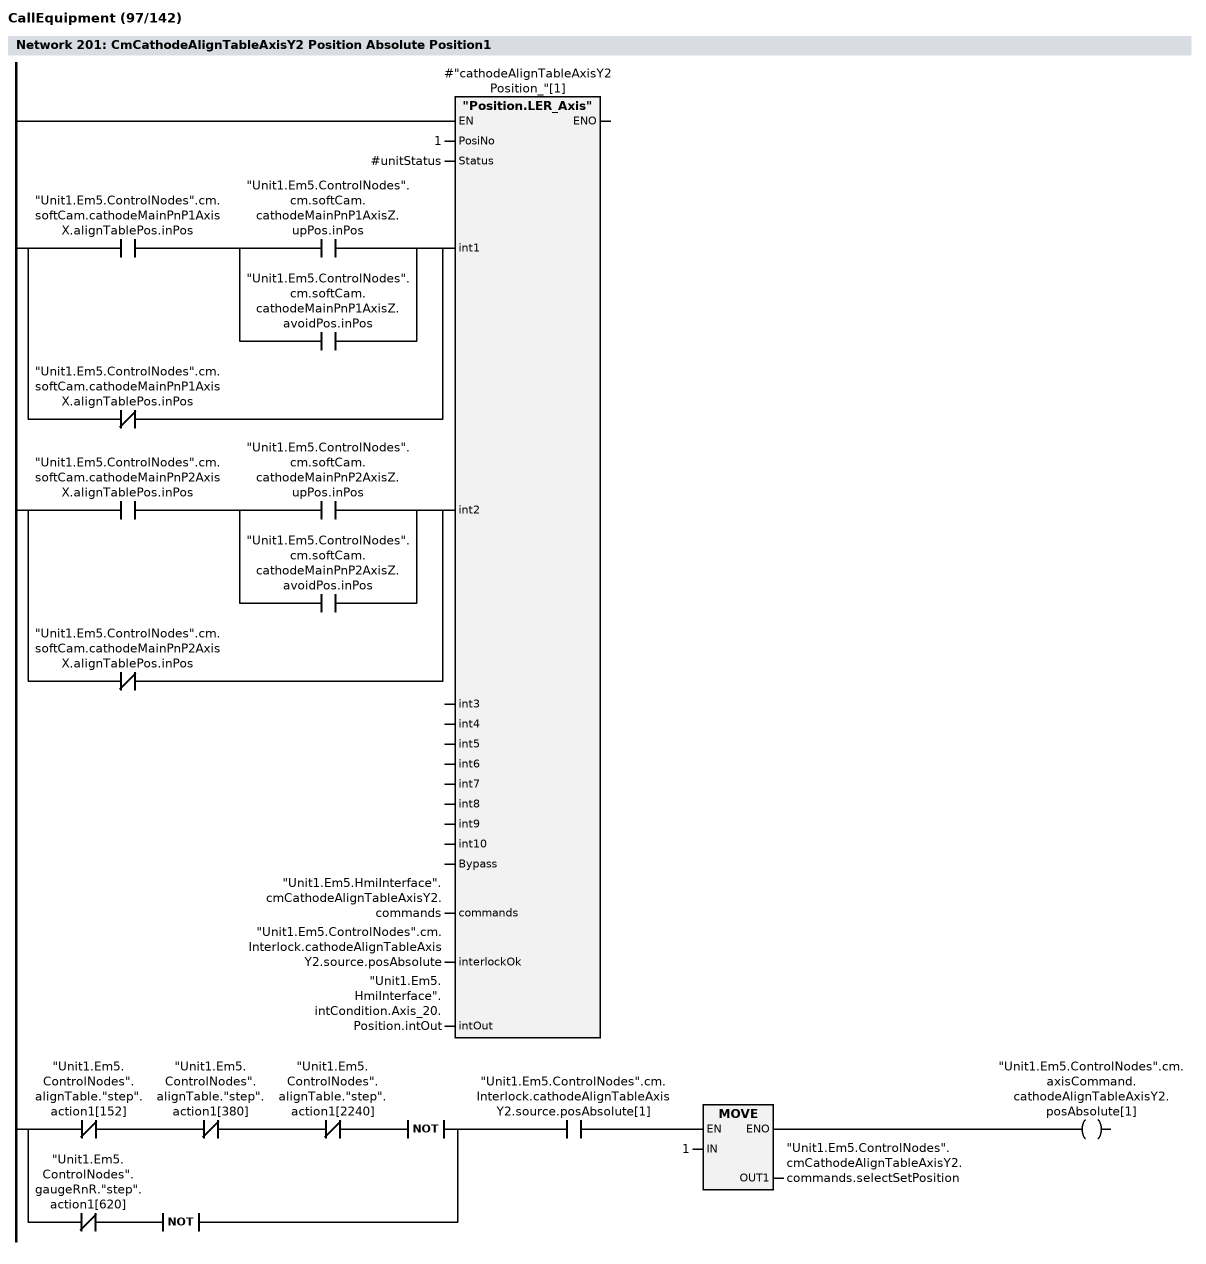
   RUNG wire#powerrail
      #"cathodeAlignTableAxisY2 Position_"[1](int1 := wire#w2, int2 := wire#w4, PosiNo := 1, Status := #unitStatus, int3 :=, int4 :=, int5 :=, int6 :=, int7 :=, int8 :=, int9 :=, int10 :=, Bypass :=, commands := "Unit1.Em5.HmiInterface".cmCathodeAlignTableAxisY2.commands, interlockOk := "Unit1.Em5.ControlNodes".cm.Interlock.cathodeAlignTableAxisY2.source.posAbsolute, intOut := "Unit1.Em5.HmiInterface".intCondition.Axis_20.Position.intOut)
   END_RUNG
   RUNG wire#powerrail
      Contact( "Unit1.Em5.ControlNodes".cm.softCam.cathodeMainPnP1AxisX.alignTablePos.inPos )
      wire#w1
      Contact( "Unit1.Em5.ControlNodes".cm.softCam.cathodeMainPnP1AxisZ.upPos.inPos )
   END_RUNG wire#w2
   RUNG wire#w1
      Contact( "Unit1.Em5.ControlNodes".cm.softCam.cathodeMainPnP1AxisZ.avoidPos.inPos )
   END_RUNG wire#w2
   RUNG wire#powerrail
      I_Contact( "Unit1.Em5.ControlNodes".cm.softCam.cathodeMainPnP1AxisX.alignTablePos.inPos )
   END_RUNG wire#w2
   RUNG wire#powerrail
      Contact( "Unit1.Em5.ControlNodes".cm.softCam.cathodeMainPnP2AxisX.alignTablePos.inPos )
      wire#w3
      Contact( "Unit1.Em5.ControlNodes".cm.softCam.cathodeMainPnP2AxisZ.upPos.inPos )
   END_RUNG wire#w4
   RUNG wire#w3
      Contact( "Unit1.Em5.ControlNodes".cm.softCam.cathodeMainPnP2AxisZ.avoidPos.inPos )
   END_RUNG wire#w4
   RUNG wire#powerrail
      I_Contact( "Unit1.Em5.ControlNodes".cm.softCam.cathodeMainPnP2AxisX.alignTablePos.inPos )
   END_RUNG wire#w4
   RUNG wire#powerrail
      I_Contact( "Unit1.Em5.ControlNodes".alignTable."step".action1[152] )
      I_Contact( "Unit1.Em5.ControlNodes".alignTable."step".action1[380] )
      I_Contact( "Unit1.Em5.ControlNodes".alignTable."step".action1[2240] )
      Not()
      wire#w5
      Contact( "Unit1.Em5.ControlNodes".cm.Interlock.cathodeAlignTableAxisY2.source.posAbsolute[1] )
      Move(in := 1, out1 => "Unit1.Em5.ControlNodes".cmCathodeAlignTableAxisY2.commands.selectSetPosition)
      Coil( "Unit1.Em5.ControlNodes".cm.axisCommand.cathodeAlignTableAxisY2.posAbsolute[1] )
   END_RUNG
   RUNG wire#powerrail
      I_Contact( "Unit1.Em5.ControlNodes".gaugeRnR."step".action1[620] )
      Not()
   END_RUNG wire#w5
   // the same network as SCL:
   #"cathodeAlignTableAxisY2 Position_"[1](PosiNo := 1,   // "Position.LER_Axis"
                           Status := #unitStatus,
                           int1 := ("Unit1.Em5.ControlNodes".cm.softCam.cathodeMainPnP1AxisX.alignTablePos.inPos AND ("Unit1.Em5.ControlNodes".cm.softCam.cathodeMainPnP1AxisZ.upPos.inPos OR "Unit1.Em5.ControlNodes".cm.softCam.cathodeMainPnP1AxisZ.avoidPos.inPos)) OR NOT "Unit1.Em5.ControlNodes".cm.softCam.cathodeMainPnP1AxisX.alignTablePos.inPos,
                           int2 := ("Unit1.Em5.ControlNodes".cm.softCam.cathodeMainPnP2AxisX.alignTablePos.inPos AND ("Unit1.Em5.ControlNodes".cm.softCam.cathodeMainPnP2AxisZ.upPos.inPos OR "Unit1.Em5.ControlNodes".cm.softCam.cathodeMainPnP2AxisZ.avoidPos.inPos)) OR NOT "Unit1.Em5.ControlNodes".cm.softCam.cathodeMainPnP2AxisX.alignTablePos.inPos,
                           commands := "Unit1.Em5.HmiInterface".cmCathodeAlignTableAxisY2.commands,
                           interlockOk := "Unit1.Em5.ControlNodes".cm.Interlock.cathodeAlignTableAxisY2.source.posAbsolute,
                           intOut := "Unit1.Em5.HmiInterface".intCondition.Axis_20.Position.intOut);
   #_w1 := (NOT (NOT "Unit1.Em5.ControlNodes".alignTable."step".action1[152] AND NOT "Unit1.Em5.ControlNodes".alignTable."step".action1[380] AND NOT "Unit1.Em5.ControlNodes".alignTable."step".action1[2240]) OR NOT (NOT "Unit1.Em5.ControlNodes".gaugeRnR."step".action1[620])) AND "Unit1.Em5.ControlNodes".cm.Interlock.cathodeAlignTableAxisY2.source.posAbsolute[1];
   IF #_w1 THEN "Unit1.Em5.ControlNodes".cmCathodeAlignTableAxisY2.commands.selectSetPosition := 1; END_IF;
   "Unit1.Em5.ControlNodes".cm.axisCommand.cathodeAlignTableAxisY2.posAbsolute[1] := #_w1;
END_REGION

REGION Network 202: CmCathodeAlignTableAxisY2 Position Absolute Position2
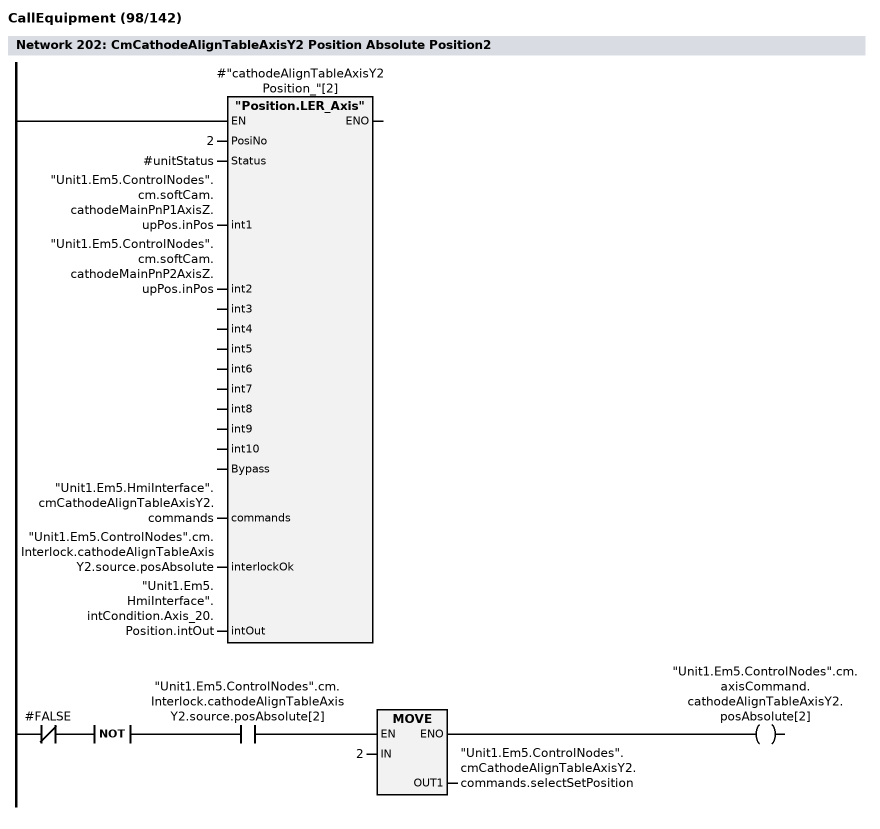
   RUNG wire#powerrail
      #"cathodeAlignTableAxisY2 Position_"[2](PosiNo := 2, Status := #unitStatus, int1 := "Unit1.Em5.ControlNodes".cm.softCam.cathodeMainPnP1AxisZ.upPos.inPos, int2 := "Unit1.Em5.ControlNodes".cm.softCam.cathodeMainPnP2AxisZ.upPos.inPos, int3 :=, int4 :=, int5 :=, int6 :=, int7 :=, int8 :=, int9 :=, int10 :=, Bypass :=, commands := "Unit1.Em5.HmiInterface".cmCathodeAlignTableAxisY2.commands, interlockOk := "Unit1.Em5.ControlNodes".cm.Interlock.cathodeAlignTableAxisY2.source.posAbsolute, intOut := "Unit1.Em5.HmiInterface".intCondition.Axis_20.Position.intOut)
   END_RUNG
   RUNG wire#powerrail
      I_Contact( #FALSE )
      Not()
      Contact( "Unit1.Em5.ControlNodes".cm.Interlock.cathodeAlignTableAxisY2.source.posAbsolute[2] )
      Move(in := 2, out1 => "Unit1.Em5.ControlNodes".cmCathodeAlignTableAxisY2.commands.selectSetPosition)
      Coil( "Unit1.Em5.ControlNodes".cm.axisCommand.cathodeAlignTableAxisY2.posAbsolute[2] )
   END_RUNG
   // the same network as SCL:
   #"cathodeAlignTableAxisY2 Position_"[2](PosiNo := 2,   // "Position.LER_Axis"
                           Status := #unitStatus,
                           int1 := "Unit1.Em5.ControlNodes".cm.softCam.cathodeMainPnP1AxisZ.upPos.inPos,
                           int2 := "Unit1.Em5.ControlNodes".cm.softCam.cathodeMainPnP2AxisZ.upPos.inPos,
                           commands := "Unit1.Em5.HmiInterface".cmCathodeAlignTableAxisY2.commands,
                           interlockOk := "Unit1.Em5.ControlNodes".cm.Interlock.cathodeAlignTableAxisY2.source.posAbsolute,
                           intOut := "Unit1.Em5.HmiInterface".intCondition.Axis_20.Position.intOut);
   #_w1 := NOT (NOT #FALSE) AND "Unit1.Em5.ControlNodes".cm.Interlock.cathodeAlignTableAxisY2.source.posAbsolute[2];
   IF #_w1 THEN "Unit1.Em5.ControlNodes".cmCathodeAlignTableAxisY2.commands.selectSetPosition := 2; END_IF;
   "Unit1.Em5.ControlNodes".cm.axisCommand.cathodeAlignTableAxisY2.posAbsolute[2] := #_w1;
END_REGION

REGION Network 203: CmCathodeAlignTableAxisY2 Position Absolute Position3
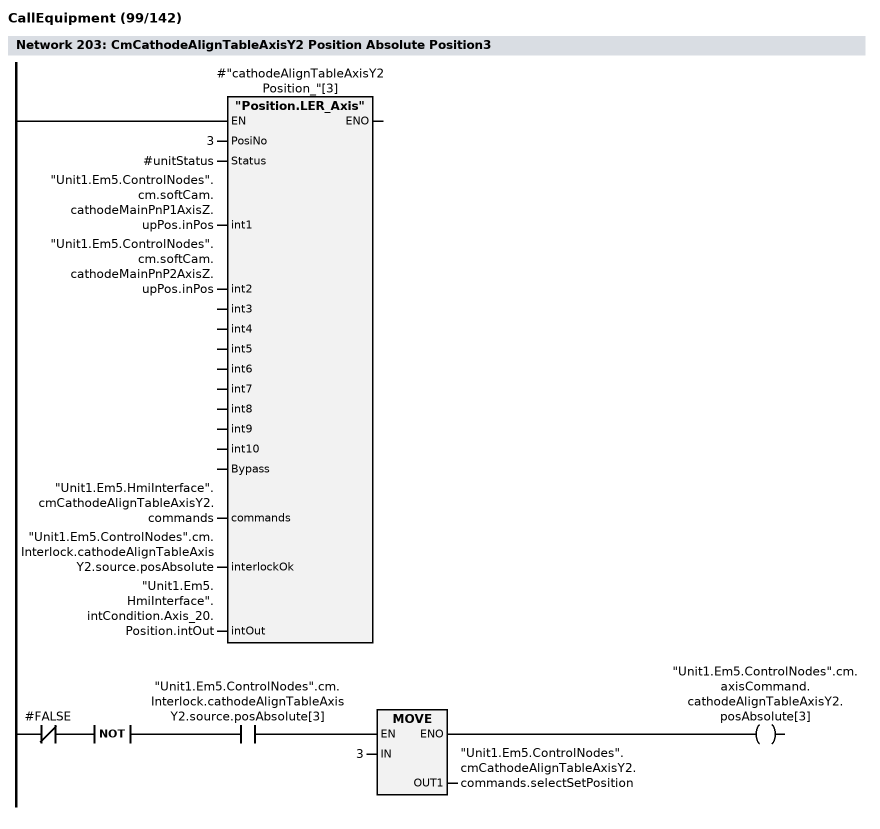
   RUNG wire#powerrail
      #"cathodeAlignTableAxisY2 Position_"[3](PosiNo := 3, Status := #unitStatus, int1 := "Unit1.Em5.ControlNodes".cm.softCam.cathodeMainPnP1AxisZ.upPos.inPos, int2 := "Unit1.Em5.ControlNodes".cm.softCam.cathodeMainPnP2AxisZ.upPos.inPos, int3 :=, int4 :=, int5 :=, int6 :=, int7 :=, int8 :=, int9 :=, int10 :=, Bypass :=, commands := "Unit1.Em5.HmiInterface".cmCathodeAlignTableAxisY2.commands, interlockOk := "Unit1.Em5.ControlNodes".cm.Interlock.cathodeAlignTableAxisY2.source.posAbsolute, intOut := "Unit1.Em5.HmiInterface".intCondition.Axis_20.Position.intOut)
   END_RUNG
   RUNG wire#powerrail
      I_Contact( #FALSE )
      Not()
      Contact( "Unit1.Em5.ControlNodes".cm.Interlock.cathodeAlignTableAxisY2.source.posAbsolute[3] )
      Move(in := 3, out1 => "Unit1.Em5.ControlNodes".cmCathodeAlignTableAxisY2.commands.selectSetPosition)
      Coil( "Unit1.Em5.ControlNodes".cm.axisCommand.cathodeAlignTableAxisY2.posAbsolute[3] )
   END_RUNG
   // the same network as SCL:
   #"cathodeAlignTableAxisY2 Position_"[3](PosiNo := 3,   // "Position.LER_Axis"
                           Status := #unitStatus,
                           int1 := "Unit1.Em5.ControlNodes".cm.softCam.cathodeMainPnP1AxisZ.upPos.inPos,
                           int2 := "Unit1.Em5.ControlNodes".cm.softCam.cathodeMainPnP2AxisZ.upPos.inPos,
                           commands := "Unit1.Em5.HmiInterface".cmCathodeAlignTableAxisY2.commands,
                           interlockOk := "Unit1.Em5.ControlNodes".cm.Interlock.cathodeAlignTableAxisY2.source.posAbsolute,
                           intOut := "Unit1.Em5.HmiInterface".intCondition.Axis_20.Position.intOut);
   #_w1 := NOT (NOT #FALSE) AND "Unit1.Em5.ControlNodes".cm.Interlock.cathodeAlignTableAxisY2.source.posAbsolute[3];
   IF #_w1 THEN "Unit1.Em5.ControlNodes".cmCathodeAlignTableAxisY2.commands.selectSetPosition := 3; END_IF;
   "Unit1.Em5.ControlNodes".cm.axisCommand.cathodeAlignTableAxisY2.posAbsolute[3] := #_w1;
END_REGION

REGION Network 204: CmCathodeAlignTableAxisY2 Position Absolute Position4
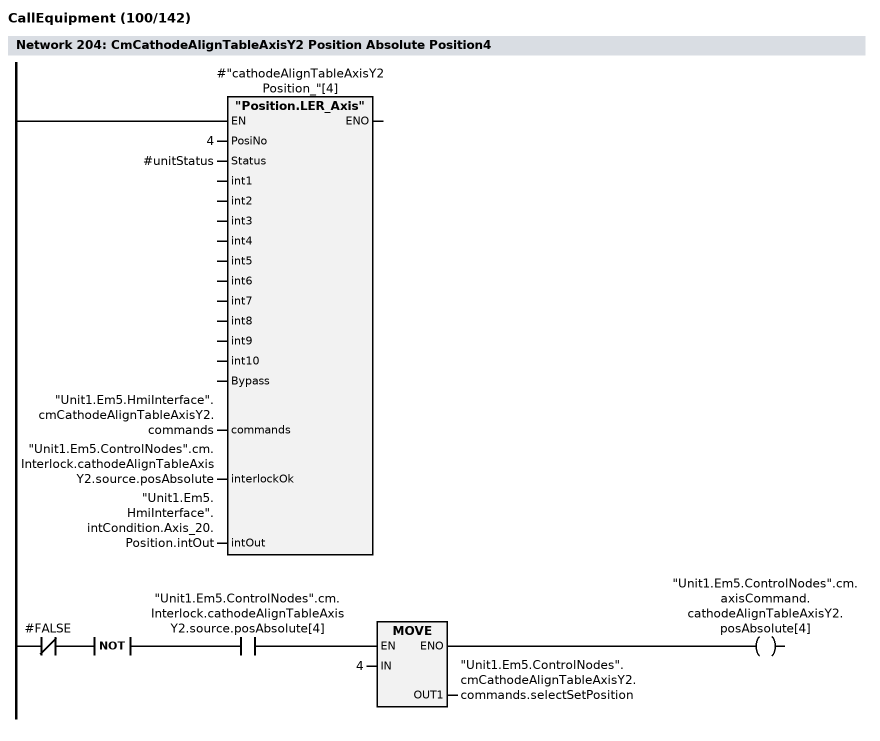
   RUNG wire#powerrail
      #"cathodeAlignTableAxisY2 Position_"[4](PosiNo := 4, Status := #unitStatus, int1 :=, int2 :=, int3 :=, int4 :=, int5 :=, int6 :=, int7 :=, int8 :=, int9 :=, int10 :=, Bypass :=, commands := "Unit1.Em5.HmiInterface".cmCathodeAlignTableAxisY2.commands, interlockOk := "Unit1.Em5.ControlNodes".cm.Interlock.cathodeAlignTableAxisY2.source.posAbsolute, intOut := "Unit1.Em5.HmiInterface".intCondition.Axis_20.Position.intOut)
   END_RUNG
   RUNG wire#powerrail
      I_Contact( #FALSE )
      Not()
      Contact( "Unit1.Em5.ControlNodes".cm.Interlock.cathodeAlignTableAxisY2.source.posAbsolute[4] )
      Move(in := 4, out1 => "Unit1.Em5.ControlNodes".cmCathodeAlignTableAxisY2.commands.selectSetPosition)
      Coil( "Unit1.Em5.ControlNodes".cm.axisCommand.cathodeAlignTableAxisY2.posAbsolute[4] )
   END_RUNG
   // the same network as SCL:
   #"cathodeAlignTableAxisY2 Position_"[4](PosiNo := 4,   // "Position.LER_Axis"
                           Status := #unitStatus,
                           commands := "Unit1.Em5.HmiInterface".cmCathodeAlignTableAxisY2.commands,
                           interlockOk := "Unit1.Em5.ControlNodes".cm.Interlock.cathodeAlignTableAxisY2.source.posAbsolute,
                           intOut := "Unit1.Em5.HmiInterface".intCondition.Axis_20.Position.intOut);
   #_w1 := NOT (NOT #FALSE) AND "Unit1.Em5.ControlNodes".cm.Interlock.cathodeAlignTableAxisY2.source.posAbsolute[4];
   IF #_w1 THEN "Unit1.Em5.ControlNodes".cmCathodeAlignTableAxisY2.commands.selectSetPosition := 4; END_IF;
   "Unit1.Em5.ControlNodes".cm.axisCommand.cathodeAlignTableAxisY2.posAbsolute[4] := #_w1;
END_REGION

REGION Network 205: CmCathodeAlignTableAxisY2 Position Absolute Position5
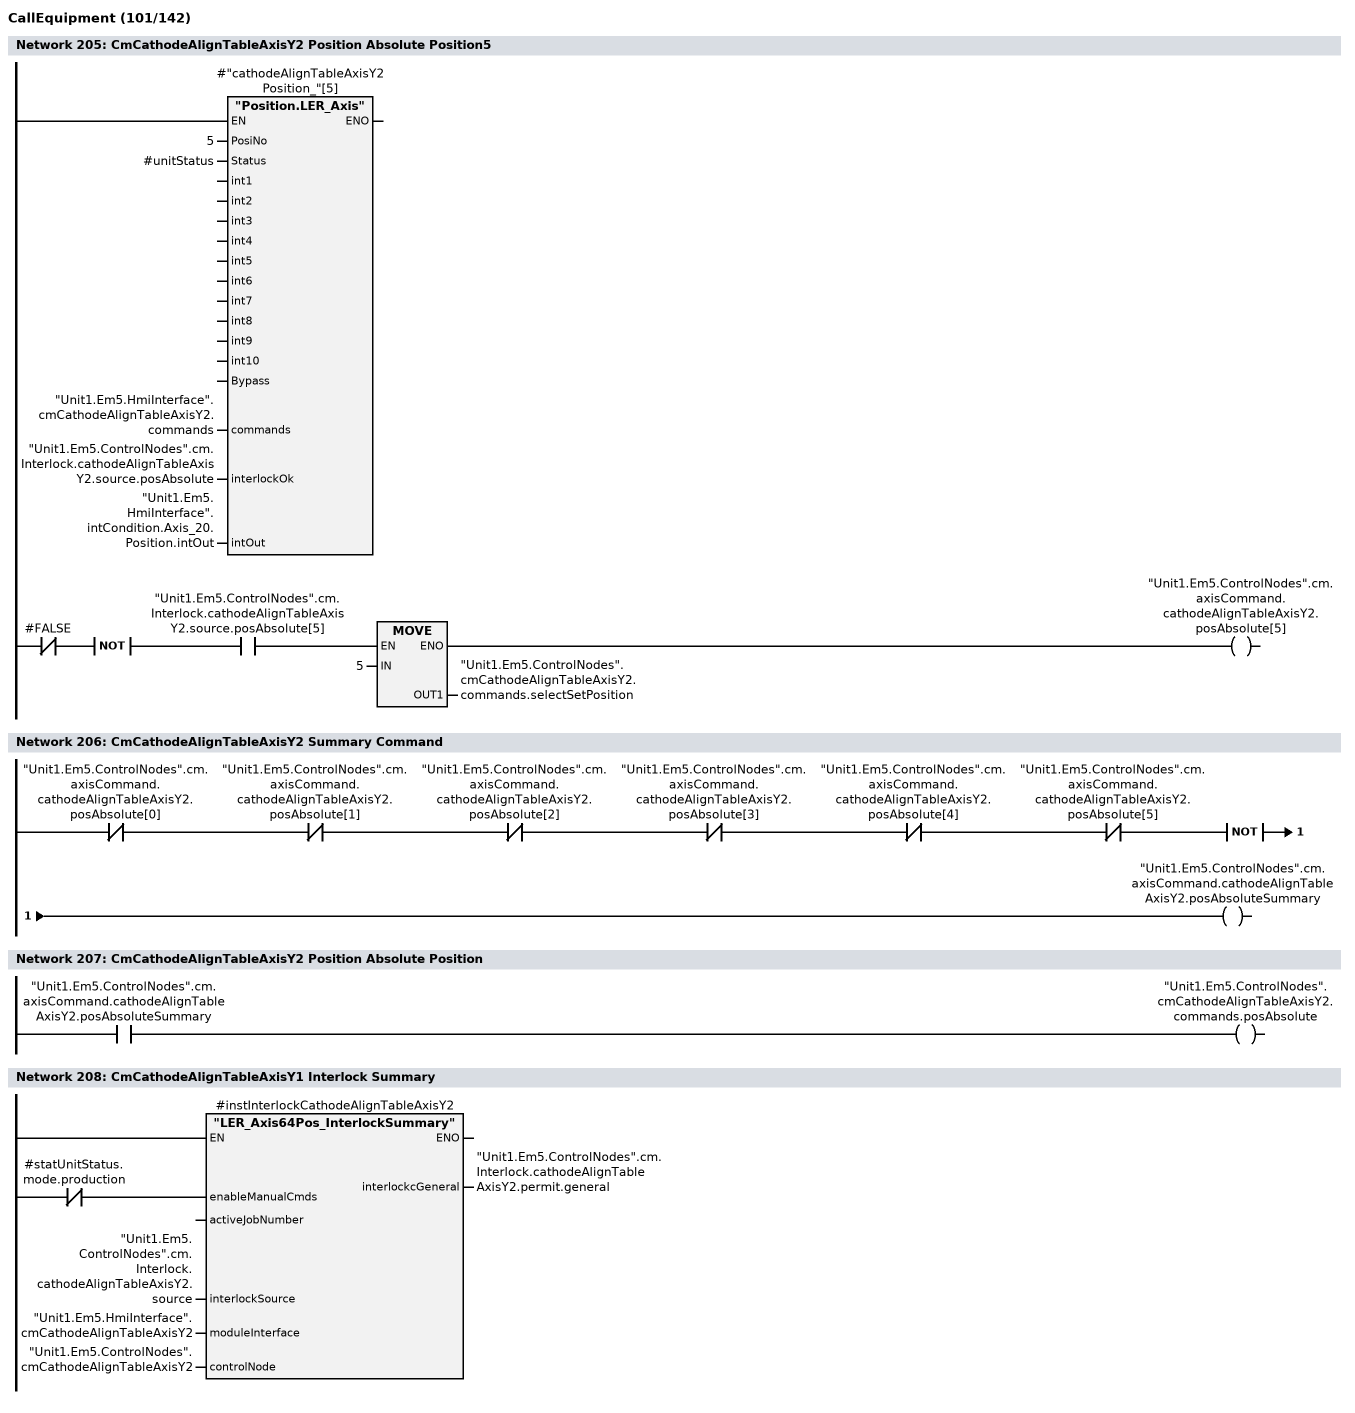
   RUNG wire#powerrail
      #"cathodeAlignTableAxisY2 Position_"[5](PosiNo := 5, Status := #unitStatus, int1 :=, int2 :=, int3 :=, int4 :=, int5 :=, int6 :=, int7 :=, int8 :=, int9 :=, int10 :=, Bypass :=, commands := "Unit1.Em5.HmiInterface".cmCathodeAlignTableAxisY2.commands, interlockOk := "Unit1.Em5.ControlNodes".cm.Interlock.cathodeAlignTableAxisY2.source.posAbsolute, intOut := "Unit1.Em5.HmiInterface".intCondition.Axis_20.Position.intOut)
   END_RUNG
   RUNG wire#powerrail
      I_Contact( #FALSE )
      Not()
      Contact( "Unit1.Em5.ControlNodes".cm.Interlock.cathodeAlignTableAxisY2.source.posAbsolute[5] )
      Move(in := 5, out1 => "Unit1.Em5.ControlNodes".cmCathodeAlignTableAxisY2.commands.selectSetPosition)
      Coil( "Unit1.Em5.ControlNodes".cm.axisCommand.cathodeAlignTableAxisY2.posAbsolute[5] )
   END_RUNG
   // the same network as SCL:
   #"cathodeAlignTableAxisY2 Position_"[5](PosiNo := 5,   // "Position.LER_Axis"
                           Status := #unitStatus,
                           commands := "Unit1.Em5.HmiInterface".cmCathodeAlignTableAxisY2.commands,
                           interlockOk := "Unit1.Em5.ControlNodes".cm.Interlock.cathodeAlignTableAxisY2.source.posAbsolute,
                           intOut := "Unit1.Em5.HmiInterface".intCondition.Axis_20.Position.intOut);
   #_w1 := NOT (NOT #FALSE) AND "Unit1.Em5.ControlNodes".cm.Interlock.cathodeAlignTableAxisY2.source.posAbsolute[5];
   IF #_w1 THEN "Unit1.Em5.ControlNodes".cmCathodeAlignTableAxisY2.commands.selectSetPosition := 5; END_IF;
   "Unit1.Em5.ControlNodes".cm.axisCommand.cathodeAlignTableAxisY2.posAbsolute[5] := #_w1;
END_REGION

REGION Network 206: CmCathodeAlignTableAxisY2 Summary Command
   RUNG wire#powerrail
      I_Contact( "Unit1.Em5.ControlNodes".cm.axisCommand.cathodeAlignTableAxisY2.posAbsolute[0] )
      I_Contact( "Unit1.Em5.ControlNodes".cm.axisCommand.cathodeAlignTableAxisY2.posAbsolute[1] )
      I_Contact( "Unit1.Em5.ControlNodes".cm.axisCommand.cathodeAlignTableAxisY2.posAbsolute[2] )
      I_Contact( "Unit1.Em5.ControlNodes".cm.axisCommand.cathodeAlignTableAxisY2.posAbsolute[3] )
      I_Contact( "Unit1.Em5.ControlNodes".cm.axisCommand.cathodeAlignTableAxisY2.posAbsolute[4] )
      I_Contact( "Unit1.Em5.ControlNodes".cm.axisCommand.cathodeAlignTableAxisY2.posAbsolute[5] )
      Not()
      Coil( "Unit1.Em5.ControlNodes".cm.axisCommand.cathodeAlignTableAxisY2.posAbsoluteSummary )
   END_RUNG
   // the same network as SCL:
   "Unit1.Em5.ControlNodes".cm.axisCommand.cathodeAlignTableAxisY2.posAbsoluteSummary := NOT (NOT "Unit1.Em5.ControlNodes".cm.axisCommand.cathodeAlignTableAxisY2.posAbsolute[0] AND NOT "Unit1.Em5.ControlNodes".cm.axisCommand.cathodeAlignTableAxisY2.posAbsolute[1] AND NOT "Unit1.Em5.ControlNodes".cm.axisCommand.cathodeAlignTableAxisY2.posAbsolute[2] AND NOT "Unit1.Em5.ControlNodes".cm.axisCommand.cathodeAlignTableAxisY2.posAbsolute[3] AND NOT "Unit1.Em5.ControlNodes".cm.axisCommand.cathodeAlignTableAxisY2.posAbsolute[4] AND NOT "Unit1.Em5.ControlNodes".cm.axisCommand.cathodeAlignTableAxisY2.posAbsolute[5]);
END_REGION

REGION Network 207: CmCathodeAlignTableAxisY2 Position Absolute Position
   RUNG wire#powerrail
      Contact( "Unit1.Em5.ControlNodes".cm.axisCommand.cathodeAlignTableAxisY2.posAbsoluteSummary )
      Coil( "Unit1.Em5.ControlNodes".cmCathodeAlignTableAxisY2.commands.posAbsolute )
   END_RUNG
   // the same network as SCL:
   "Unit1.Em5.ControlNodes".cmCathodeAlignTableAxisY2.commands.posAbsolute := "Unit1.Em5.ControlNodes".cm.axisCommand.cathodeAlignTableAxisY2.posAbsoluteSummary;
END_REGION

REGION Network 208: CmCathodeAlignTableAxisY1 Interlock Summary
   RUNG wire#powerrail
      #instInterlockCathodeAlignTableAxisY2(enableManualCmds := wire#w1, activeJobNumber :=, interlockSource := "Unit1.Em5.ControlNodes".cm.Interlock.cathodeAlignTableAxisY2.source, moduleInterface := "Unit1.Em5.HmiInterface".cmCathodeAlignTableAxisY2, controlNode := "Unit1.Em5.ControlNodes".cmCathodeAlignTableAxisY2, interlockcGeneral => "Unit1.Em5.ControlNodes".cm.Interlock.cathodeAlignTableAxisY2.permit.general)
   END_RUNG
   RUNG wire#powerrail
      I_Contact( #statUnitStatus.mode.production )
   END_RUNG wire#w1
   // the same network as SCL:
   #instInterlockCathodeAlignTableAxisY2(enableManualCmds := NOT #statUnitStatus.mode.production,   // "LER_Axis64Pos_InterlockSummary"
                           interlockSource := "Unit1.Em5.ControlNodes".cm.Interlock.cathodeAlignTableAxisY2.source,
                           moduleInterface := "Unit1.Em5.HmiInterface".cmCathodeAlignTableAxisY2,
                           controlNode := "Unit1.Em5.ControlNodes".cmCathodeAlignTableAxisY2,
                           interlockcGeneral => "Unit1.Em5.ControlNodes".cm.Interlock.cathodeAlignTableAxisY2.permit.general);
END_REGION

REGION Network 209: CmCathodeAlignTableAxisY2 velocity/speed
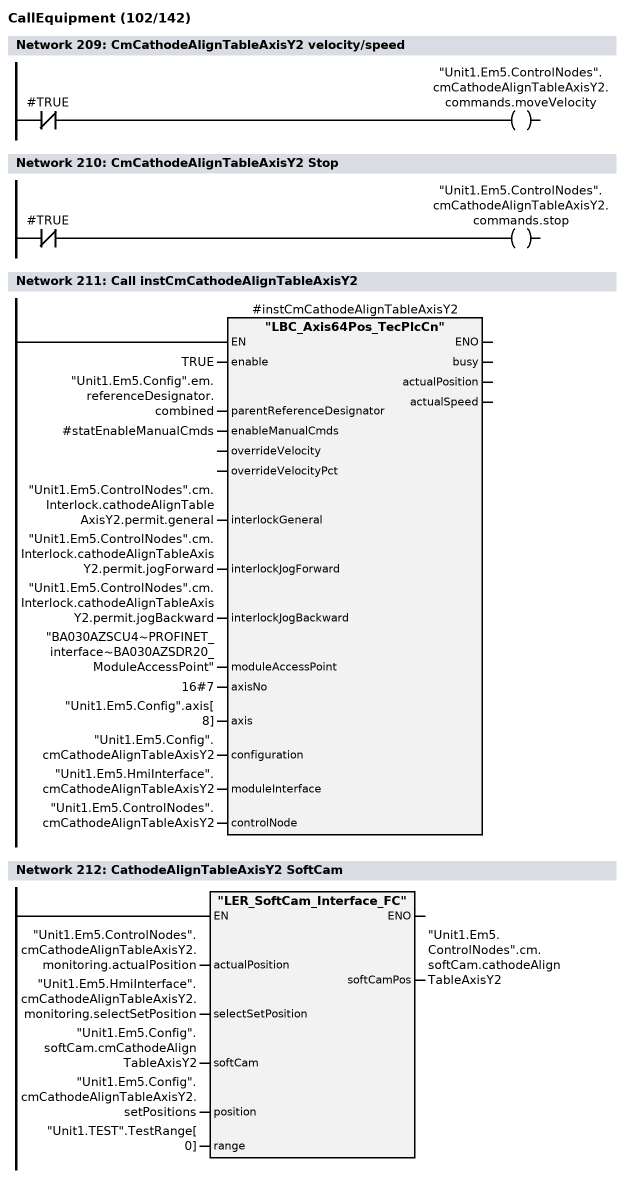
   RUNG wire#powerrail
      I_Contact( #TRUE )
      Coil( "Unit1.Em5.ControlNodes".cmCathodeAlignTableAxisY2.commands.moveVelocity )
   END_RUNG
   // the same network as SCL:
   "Unit1.Em5.ControlNodes".cmCathodeAlignTableAxisY2.commands.moveVelocity := NOT #TRUE;
END_REGION

REGION Network 210: CmCathodeAlignTableAxisY2 Stop
   RUNG wire#powerrail
      I_Contact( #TRUE )
      Coil( "Unit1.Em5.ControlNodes".cmCathodeAlignTableAxisY2.commands.stop )
   END_RUNG
   // the same network as SCL:
   "Unit1.Em5.ControlNodes".cmCathodeAlignTableAxisY2.commands.stop := NOT #TRUE;
END_REGION

REGION Network 211: Call instCmCathodeAlignTableAxisY2
   RUNG wire#powerrail
      #instCmCathodeAlignTableAxisY2(enable := TRUE, parentReferenceDesignator := "Unit1.Em5.Config".em.referenceDesignator.combined, enableManualCmds := #statEnableManualCmds, overrideVelocity :=, overrideVelocityPct :=, interlockGeneral := "Unit1.Em5.ControlNodes".cm.Interlock.cathodeAlignTableAxisY2.permit.general, interlockJogForward := "Unit1.Em5.ControlNodes".cm.Interlock.cathodeAlignTableAxisY2.permit.jogForward, interlockJogBackward := "Unit1.Em5.ControlNodes".cm.Interlock.cathodeAlignTableAxisY2.permit.jogBackward, moduleAccessPoint := "BA030AZSCU4~PROFINET_interface~BA030AZSDR20_ModuleAccessPoint", axisNo := 16#7, axis := "Unit1.Em5.Config".axis[8], configuration := "Unit1.Em5.Config".cmCathodeAlignTableAxisY2, moduleInterface := "Unit1.Em5.HmiInterface".cmCathodeAlignTableAxisY2, controlNode := "Unit1.Em5.ControlNodes".cmCathodeAlignTableAxisY2, busy =>, actualPosition =>, actualSpeed =>)
   END_RUNG
   // the same network as SCL:
   #instCmCathodeAlignTableAxisY2(enable := TRUE,   // "LBC_Axis64Pos_TecPlcCn"
                           parentReferenceDesignator := "Unit1.Em5.Config".em.referenceDesignator.combined,
                           enableManualCmds := #statEnableManualCmds,
                           interlockGeneral := "Unit1.Em5.ControlNodes".cm.Interlock.cathodeAlignTableAxisY2.permit.general,
                           interlockJogForward := "Unit1.Em5.ControlNodes".cm.Interlock.cathodeAlignTableAxisY2.permit.jogForward,
                           interlockJogBackward := "Unit1.Em5.ControlNodes".cm.Interlock.cathodeAlignTableAxisY2.permit.jogBackward,
                           moduleAccessPoint := "BA030AZSCU4~PROFINET_interface~BA030AZSDR20_ModuleAccessPoint",
                           axisNo := 16#7,
                           axis := "Unit1.Em5.Config".axis[8],
                           configuration := "Unit1.Em5.Config".cmCathodeAlignTableAxisY2,
                           moduleInterface := "Unit1.Em5.HmiInterface".cmCathodeAlignTableAxisY2,
                           controlNode := "Unit1.Em5.ControlNodes".cmCathodeAlignTableAxisY2);
END_REGION

REGION Network 212: CathodeAlignTableAxisY2 SoftCam
   RUNG wire#powerrail
      "LER_SoftCam_Interface_FC"(actualPosition := "Unit1.Em5.ControlNodes".cmCathodeAlignTableAxisY2.monitoring.actualPosition, selectSetPosition := "Unit1.Em5.HmiInterface".cmCathodeAlignTableAxisY2.monitoring.selectSetPosition, softCam := "Unit1.Em5.Config".softCam.cmCathodeAlignTableAxisY2, position := "Unit1.Em5.Config".cmCathodeAlignTableAxisY2.setPositions, range := "Unit1.TEST".TestRange[0], softCamPos => "Unit1.Em5.ControlNodes".cm.softCam.cathodeAlignTableAxisY2)
   END_RUNG
   // the same network as SCL:
   "LER_SoftCam_Interface_FC"(actualPosition := "Unit1.Em5.ControlNodes".cmCathodeAlignTableAxisY2.monitoring.actualPosition,
                           selectSetPosition := "Unit1.Em5.HmiInterface".cmCathodeAlignTableAxisY2.monitoring.selectSetPosition,
                           softCam := "Unit1.Em5.Config".softCam.cmCathodeAlignTableAxisY2,
                           position := "Unit1.Em5.Config".cmCathodeAlignTableAxisY2.setPositions,
                           range := "Unit1.TEST".TestRange[0],
                           softCamPos => "Unit1.Em5.ControlNodes".cm.softCam.cathodeAlignTableAxisY2);
END_REGION

REGION Network 213: ******************** Brake Test (Axis) ********************
END_REGION

REGION Network 214: Cathode Main PnP 1 Z-Axis Brake Test
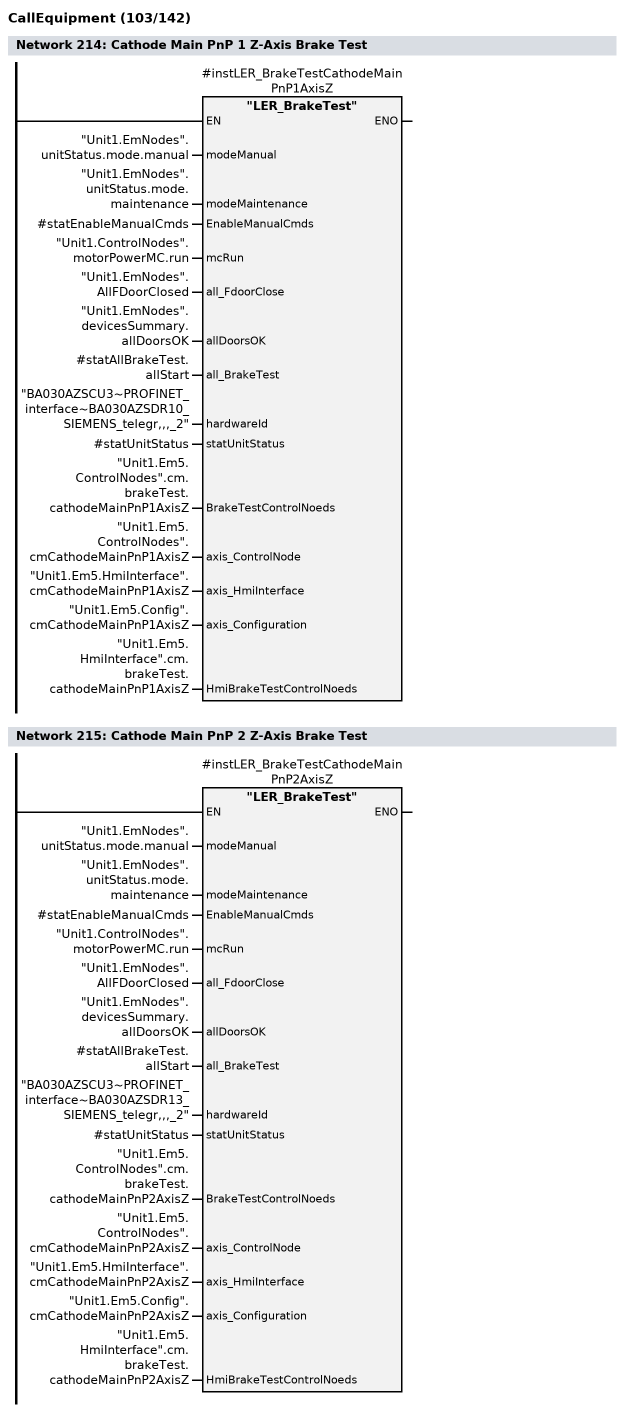
   RUNG wire#powerrail
      #instLER_BrakeTestCathodeMainPnP1AxisZ(modeManual := "Unit1.EmNodes".unitStatus.mode.manual, modeMaintenance := "Unit1.EmNodes".unitStatus.mode.maintenance, EnableManualCmds := #statEnableManualCmds, mcRun := "Unit1.ControlNodes".motorPowerMC.run, all_FdoorClose := "Unit1.EmNodes".AllFDoorClosed, allDoorsOK := "Unit1.EmNodes".devicesSummary.allDoorsOK, all_BrakeTest := #statAllBrakeTest.allStart, hardwareId := "BA030AZSCU3~PROFINET_interface~BA030AZSDR10_SIEMENS_telegr,,,_2", statUnitStatus := #statUnitStatus, BrakeTestControlNoeds := "Unit1.Em5.ControlNodes".cm.brakeTest.cathodeMainPnP1AxisZ, axis_ControlNode := "Unit1.Em5.ControlNodes".cmCathodeMainPnP1AxisZ, axis_HmiInterface := "Unit1.Em5.HmiInterface".cmCathodeMainPnP1AxisZ, axis_Configuration := "Unit1.Em5.Config".cmCathodeMainPnP1AxisZ, HmiBrakeTestControlNoeds := "Unit1.Em5.HmiInterface".cm.brakeTest.cathodeMainPnP1AxisZ)
   END_RUNG
   // the same network as SCL:
   #instLER_BrakeTestCathodeMainPnP1AxisZ(modeManual := "Unit1.EmNodes".unitStatus.mode.manual,   // "LER_BrakeTest"
                           modeMaintenance := "Unit1.EmNodes".unitStatus.mode.maintenance,
                           EnableManualCmds := #statEnableManualCmds,
                           mcRun := "Unit1.ControlNodes".motorPowerMC.run,
                           all_FdoorClose := "Unit1.EmNodes".AllFDoorClosed,
                           allDoorsOK := "Unit1.EmNodes".devicesSummary.allDoorsOK,
                           all_BrakeTest := #statAllBrakeTest.allStart,
                           hardwareId := "BA030AZSCU3~PROFINET_interface~BA030AZSDR10_SIEMENS_telegr,,,_2",
                           statUnitStatus := #statUnitStatus,
                           BrakeTestControlNoeds := "Unit1.Em5.ControlNodes".cm.brakeTest.cathodeMainPnP1AxisZ,
                           axis_ControlNode := "Unit1.Em5.ControlNodes".cmCathodeMainPnP1AxisZ,
                           axis_HmiInterface := "Unit1.Em5.HmiInterface".cmCathodeMainPnP1AxisZ,
                           axis_Configuration := "Unit1.Em5.Config".cmCathodeMainPnP1AxisZ,
                           HmiBrakeTestControlNoeds := "Unit1.Em5.HmiInterface".cm.brakeTest.cathodeMainPnP1AxisZ);
END_REGION

REGION Network 215: Cathode Main PnP 2 Z-Axis Brake Test
   RUNG wire#powerrail
      #instLER_BrakeTestCathodeMainPnP2AxisZ(modeManual := "Unit1.EmNodes".unitStatus.mode.manual, modeMaintenance := "Unit1.EmNodes".unitStatus.mode.maintenance, EnableManualCmds := #statEnableManualCmds, mcRun := "Unit1.ControlNodes".motorPowerMC.run, all_FdoorClose := "Unit1.EmNodes".AllFDoorClosed, allDoorsOK := "Unit1.EmNodes".devicesSummary.allDoorsOK, all_BrakeTest := #statAllBrakeTest.allStart, hardwareId := "BA030AZSCU3~PROFINET_interface~BA030AZSDR13_SIEMENS_telegr,,,_2", statUnitStatus := #statUnitStatus, BrakeTestControlNoeds := "Unit1.Em5.ControlNodes".cm.brakeTest.cathodeMainPnP2AxisZ, axis_ControlNode := "Unit1.Em5.ControlNodes".cmCathodeMainPnP2AxisZ, axis_HmiInterface := "Unit1.Em5.HmiInterface".cmCathodeMainPnP2AxisZ, axis_Configuration := "Unit1.Em5.Config".cmCathodeMainPnP2AxisZ, HmiBrakeTestControlNoeds := "Unit1.Em5.HmiInterface".cm.brakeTest.cathodeMainPnP2AxisZ)
   END_RUNG
   // the same network as SCL:
   #instLER_BrakeTestCathodeMainPnP2AxisZ(modeManual := "Unit1.EmNodes".unitStatus.mode.manual,   // "LER_BrakeTest"
                           modeMaintenance := "Unit1.EmNodes".unitStatus.mode.maintenance,
                           EnableManualCmds := #statEnableManualCmds,
                           mcRun := "Unit1.ControlNodes".motorPowerMC.run,
                           all_FdoorClose := "Unit1.EmNodes".AllFDoorClosed,
                           allDoorsOK := "Unit1.EmNodes".devicesSummary.allDoorsOK,
                           all_BrakeTest := #statAllBrakeTest.allStart,
                           hardwareId := "BA030AZSCU3~PROFINET_interface~BA030AZSDR13_SIEMENS_telegr,,,_2",
                           statUnitStatus := #statUnitStatus,
                           BrakeTestControlNoeds := "Unit1.Em5.ControlNodes".cm.brakeTest.cathodeMainPnP2AxisZ,
                           axis_ControlNode := "Unit1.Em5.ControlNodes".cmCathodeMainPnP2AxisZ,
                           axis_HmiInterface := "Unit1.Em5.HmiInterface".cmCathodeMainPnP2AxisZ,
                           axis_Configuration := "Unit1.Em5.Config".cmCathodeMainPnP2AxisZ,
                           HmiBrakeTestControlNoeds := "Unit1.Em5.HmiInterface".cm.brakeTest.cathodeMainPnP2AxisZ);
END_REGION

REGION Network 216: ******************** Align Table Extended Function ********************
END_REGION

REGION Network 217: Call Anode Align Table Move Calibration (LER_AlignCalibration)
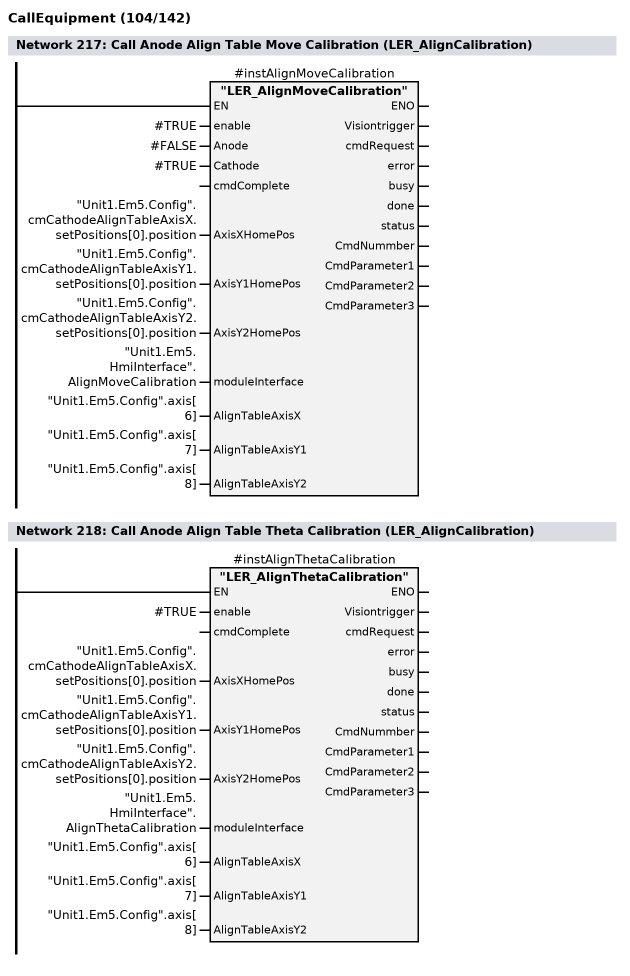
   RUNG wire#powerrail
      #instAlignMoveCalibration(enable := #TRUE, Anode := #FALSE, Cathode := #TRUE, cmdComplete :=, AxisXHomePos := "Unit1.Em5.Config".cmCathodeAlignTableAxisX.setPositions[0].position, AxisY1HomePos := "Unit1.Em5.Config".cmCathodeAlignTableAxisY1.setPositions[0].position, AxisY2HomePos := "Unit1.Em5.Config".cmCathodeAlignTableAxisY2.setPositions[0].position, moduleInterface := "Unit1.Em5.HmiInterface".AlignMoveCalibration, AlignTableAxisX := "Unit1.Em5.Config".axis[6], AlignTableAxisY1 := "Unit1.Em5.Config".axis[7], AlignTableAxisY2 := "Unit1.Em5.Config".axis[8], Visiontrigger =>, cmdRequest =>, error =>, busy =>, done =>, status =>, CmdNummber =>, CmdParameter1 =>, CmdParameter2 =>, CmdParameter3 =>)
   END_RUNG
   // the same network as SCL:
   #instAlignMoveCalibration(enable := #TRUE,   // "LER_AlignMoveCalibration"
                           Anode := #FALSE,
                           Cathode := #TRUE,
                           AxisXHomePos := "Unit1.Em5.Config".cmCathodeAlignTableAxisX.setPositions[0].position,
                           AxisY1HomePos := "Unit1.Em5.Config".cmCathodeAlignTableAxisY1.setPositions[0].position,
                           AxisY2HomePos := "Unit1.Em5.Config".cmCathodeAlignTableAxisY2.setPositions[0].position,
                           moduleInterface := "Unit1.Em5.HmiInterface".AlignMoveCalibration,
                           AlignTableAxisX := "Unit1.Em5.Config".axis[6],
                           AlignTableAxisY1 := "Unit1.Em5.Config".axis[7],
                           AlignTableAxisY2 := "Unit1.Em5.Config".axis[8]);
END_REGION

REGION Network 218: Call Anode Align Table Theta Calibration (LER_AlignCalibration)
   RUNG wire#powerrail
      #instAlignThetaCalibration(enable := #TRUE, cmdComplete :=, AxisXHomePos := "Unit1.Em5.Config".cmCathodeAlignTableAxisX.setPositions[0].position, AxisY1HomePos := "Unit1.Em5.Config".cmCathodeAlignTableAxisY1.setPositions[0].position, AxisY2HomePos := "Unit1.Em5.Config".cmCathodeAlignTableAxisY2.setPositions[0].position, moduleInterface := "Unit1.Em5.HmiInterface".AlignThetaCalibration, AlignTableAxisX := "Unit1.Em5.Config".axis[6], AlignTableAxisY1 := "Unit1.Em5.Config".axis[7], AlignTableAxisY2 := "Unit1.Em5.Config".axis[8], Visiontrigger =>, cmdRequest =>, error =>, busy =>, done =>, status =>, CmdNummber =>, CmdParameter1 =>, CmdParameter2 =>, CmdParameter3 =>)
   END_RUNG
   // the same network as SCL:
   #instAlignThetaCalibration(enable := #TRUE,   // "LER_AlignThetaCalibration"
                           AxisXHomePos := "Unit1.Em5.Config".cmCathodeAlignTableAxisX.setPositions[0].position,
                           AxisY1HomePos := "Unit1.Em5.Config".cmCathodeAlignTableAxisY1.setPositions[0].position,
                           AxisY2HomePos := "Unit1.Em5.Config".cmCathodeAlignTableAxisY2.setPositions[0].position,
                           moduleInterface := "Unit1.Em5.HmiInterface".AlignThetaCalibration,
                           AlignTableAxisX := "Unit1.Em5.Config".axis[6],
                           AlignTableAxisY1 := "Unit1.Em5.Config".axis[7],
                           AlignTableAxisY2 := "Unit1.Em5.Config".axis[8]);
END_REGION

REGION Network 219: Call Anode Align Table Y-Axis Sync Move (LER_AlignSyncMove)
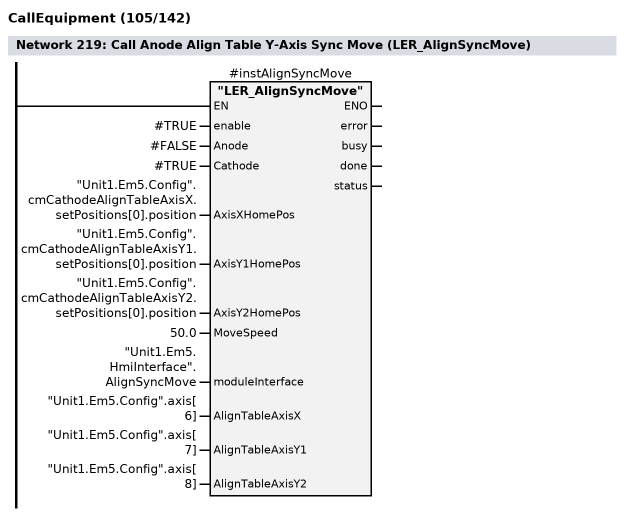
   RUNG wire#powerrail
      #instAlignSyncMove(enable := #TRUE, Anode := #FALSE, Cathode := #TRUE, AxisXHomePos := "Unit1.Em5.Config".cmCathodeAlignTableAxisX.setPositions[0].position, AxisY1HomePos := "Unit1.Em5.Config".cmCathodeAlignTableAxisY1.setPositions[0].position, AxisY2HomePos := "Unit1.Em5.Config".cmCathodeAlignTableAxisY2.setPositions[0].position, MoveSpeed := 50.0, moduleInterface := "Unit1.Em5.HmiInterface".AlignSyncMove, AlignTableAxisX := "Unit1.Em5.Config".axis[6], AlignTableAxisY1 := "Unit1.Em5.Config".axis[7], AlignTableAxisY2 := "Unit1.Em5.Config".axis[8], error =>, busy =>, done =>, status =>)
   END_RUNG
   // the same network as SCL:
   #instAlignSyncMove(enable := #TRUE,   // "LER_AlignSyncMove"
                      Anode := #FALSE,
                      Cathode := #TRUE,
                      AxisXHomePos := "Unit1.Em5.Config".cmCathodeAlignTableAxisX.setPositions[0].position,
                      AxisY1HomePos := "Unit1.Em5.Config".cmCathodeAlignTableAxisY1.setPositions[0].position,
                      AxisY2HomePos := "Unit1.Em5.Config".cmCathodeAlignTableAxisY2.setPositions[0].position,
                      MoveSpeed := 50.0,
                      moduleInterface := "Unit1.Em5.HmiInterface".AlignSyncMove,
                      AlignTableAxisX := "Unit1.Em5.Config".axis[6],
                      AlignTableAxisY1 := "Unit1.Em5.Config".axis[7],
                      AlignTableAxisY2 := "Unit1.Em5.Config".axis[8]);
END_REGION

REGION Network 220: ********** Control Modules (TwoWayActuator) **********
END_REGION

REGION Network 221: Reset CMS
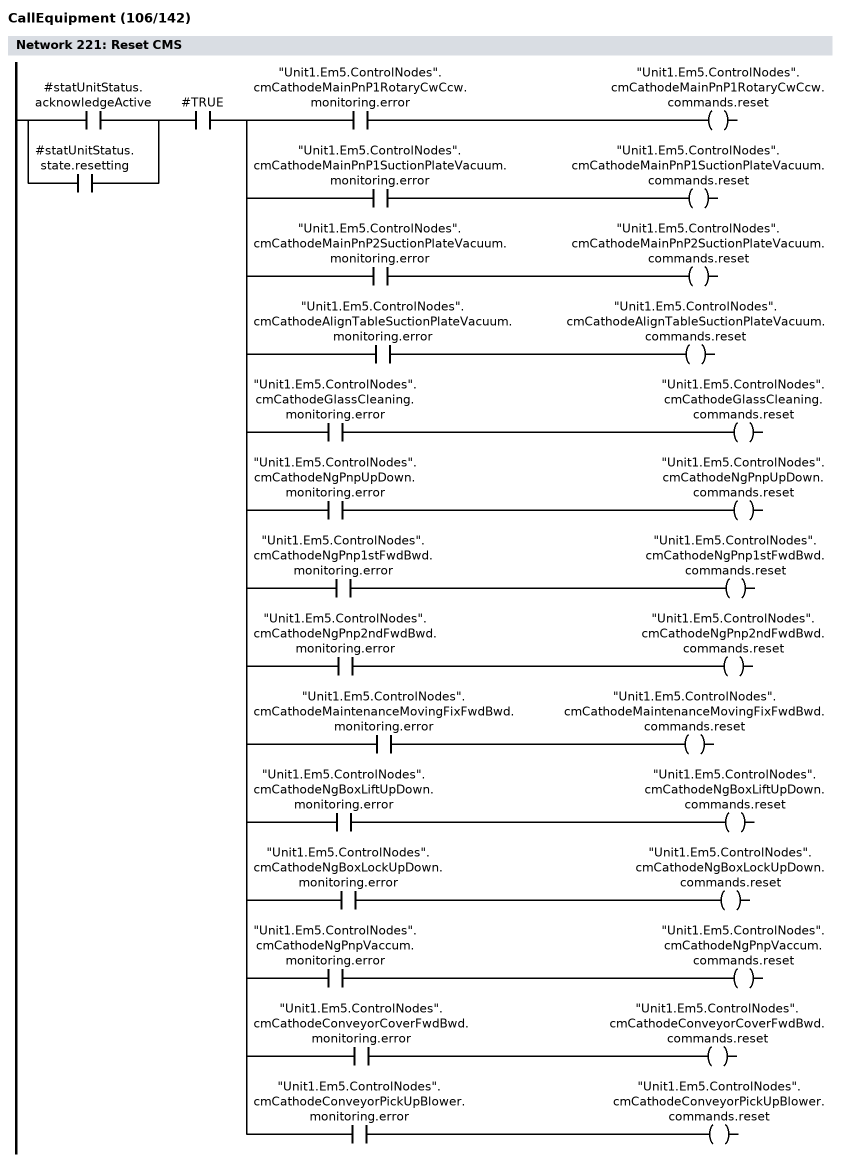
   RUNG wire#powerrail
      Contact( #statUnitStatus.acknowledgeActive )
      wire#w1
      Contact( #TRUE )
      wire#w2
      Contact( "Unit1.Em5.ControlNodes".cmCathodeMainPnP1RotaryCwCcw.monitoring.error )
      Coil( "Unit1.Em5.ControlNodes".cmCathodeMainPnP1RotaryCwCcw.commands.reset )
   END_RUNG
   RUNG wire#powerrail
      Contact( #statUnitStatus.state.resetting )
   END_RUNG wire#w1
   RUNG wire#w2
      Contact( "Unit1.Em5.ControlNodes".cmCathodeMainPnP1SuctionPlateVacuum.monitoring.error )
      Coil( "Unit1.Em5.ControlNodes".cmCathodeMainPnP1SuctionPlateVacuum.commands.reset )
   END_RUNG
   RUNG wire#w2
      Contact( "Unit1.Em5.ControlNodes".cmCathodeMainPnP2SuctionPlateVacuum.monitoring.error )
      Coil( "Unit1.Em5.ControlNodes".cmCathodeMainPnP2SuctionPlateVacuum.commands.reset )
   END_RUNG
   RUNG wire#w2
      Contact( "Unit1.Em5.ControlNodes".cmCathodeAlignTableSuctionPlateVacuum.monitoring.error )
      Coil( "Unit1.Em5.ControlNodes".cmCathodeAlignTableSuctionPlateVacuum.commands.reset )
   END_RUNG
   RUNG wire#w2
      Contact( "Unit1.Em5.ControlNodes".cmCathodeGlassCleaning.monitoring.error )
      Coil( "Unit1.Em5.ControlNodes".cmCathodeGlassCleaning.commands.reset )
   END_RUNG
   RUNG wire#w2
      Contact( "Unit1.Em5.ControlNodes".cmCathodeNgPnpUpDown.monitoring.error )
      Coil( "Unit1.Em5.ControlNodes".cmCathodeNgPnpUpDown.commands.reset )
   END_RUNG
   RUNG wire#w2
      Contact( "Unit1.Em5.ControlNodes".cmCathodeNgPnp1stFwdBwd.monitoring.error )
      Coil( "Unit1.Em5.ControlNodes".cmCathodeNgPnp1stFwdBwd.commands.reset )
   END_RUNG
   RUNG wire#w2
      Contact( "Unit1.Em5.ControlNodes".cmCathodeNgPnp2ndFwdBwd.monitoring.error )
      Coil( "Unit1.Em5.ControlNodes".cmCathodeNgPnp2ndFwdBwd.commands.reset )
   END_RUNG
   RUNG wire#w2
      Contact( "Unit1.Em5.ControlNodes".cmCathodeMaintenanceMovingFixFwdBwd.monitoring.error )
      Coil( "Unit1.Em5.ControlNodes".cmCathodeMaintenanceMovingFixFwdBwd.commands.reset )
   END_RUNG
   RUNG wire#w2
      Contact( "Unit1.Em5.ControlNodes".cmCathodeNgBoxLiftUpDown.monitoring.error )
      Coil( "Unit1.Em5.ControlNodes".cmCathodeNgBoxLiftUpDown.commands.reset )
   END_RUNG
   RUNG wire#w2
      Contact( "Unit1.Em5.ControlNodes".cmCathodeNgBoxLockUpDown.monitoring.error )
      Coil( "Unit1.Em5.ControlNodes".cmCathodeNgBoxLockUpDown.commands.reset )
   END_RUNG
   RUNG wire#w2
      Contact( "Unit1.Em5.ControlNodes".cmCathodeNgPnpVaccum.monitoring.error )
      Coil( "Unit1.Em5.ControlNodes".cmCathodeNgPnpVaccum.commands.reset )
   END_RUNG
   RUNG wire#w2
      Contact( "Unit1.Em5.ControlNodes".cmCathodeConveyorCoverFwdBwd.monitoring.error )
      Coil( "Unit1.Em5.ControlNodes".cmCathodeConveyorCoverFwdBwd.commands.reset )
   END_RUNG
   RUNG wire#w2
      Contact( "Unit1.Em5.ControlNodes".cmCathodeConveyorPickUpBlower.monitoring.error )
      Coil( "Unit1.Em5.ControlNodes".cmCathodeConveyorPickUpBlower.commands.reset )
   END_RUNG
   // the same network as SCL:
   #_w1 := (#statUnitStatus.acknowledgeActive OR #statUnitStatus.state.resetting) AND #TRUE;
   "Unit1.Em5.ControlNodes".cmCathodeMainPnP1RotaryCwCcw.commands.reset := #_w1 AND "Unit1.Em5.ControlNodes".cmCathodeMainPnP1RotaryCwCcw.monitoring.error;
   "Unit1.Em5.ControlNodes".cmCathodeMainPnP1SuctionPlateVacuum.commands.reset := #_w1 AND "Unit1.Em5.ControlNodes".cmCathodeMainPnP1SuctionPlateVacuum.monitoring.error;
   "Unit1.Em5.ControlNodes".cmCathodeMainPnP2SuctionPlateVacuum.commands.reset := #_w1 AND "Unit1.Em5.ControlNodes".cmCathodeMainPnP2SuctionPlateVacuum.monitoring.error;
   "Unit1.Em5.ControlNodes".cmCathodeAlignTableSuctionPlateVacuum.commands.reset := #_w1 AND "Unit1.Em5.ControlNodes".cmCathodeAlignTableSuctionPlateVacuum.monitoring.error;
   "Unit1.Em5.ControlNodes".cmCathodeGlassCleaning.commands.reset := #_w1 AND "Unit1.Em5.ControlNodes".cmCathodeGlassCleaning.monitoring.error;
   "Unit1.Em5.ControlNodes".cmCathodeNgPnpUpDown.commands.reset := #_w1 AND "Unit1.Em5.ControlNodes".cmCathodeNgPnpUpDown.monitoring.error;
   "Unit1.Em5.ControlNodes".cmCathodeNgPnp1stFwdBwd.commands.reset := #_w1 AND "Unit1.Em5.ControlNodes".cmCathodeNgPnp1stFwdBwd.monitoring.error;
   "Unit1.Em5.ControlNodes".cmCathodeNgPnp2ndFwdBwd.commands.reset := #_w1 AND "Unit1.Em5.ControlNodes".cmCathodeNgPnp2ndFwdBwd.monitoring.error;
   "Unit1.Em5.ControlNodes".cmCathodeMaintenanceMovingFixFwdBwd.commands.reset := #_w1 AND "Unit1.Em5.ControlNodes".cmCathodeMaintenanceMovingFixFwdBwd.monitoring.error;
   "Unit1.Em5.ControlNodes".cmCathodeNgBoxLiftUpDown.commands.reset := #_w1 AND "Unit1.Em5.ControlNodes".cmCathodeNgBoxLiftUpDown.monitoring.error;
   "Unit1.Em5.ControlNodes".cmCathodeNgBoxLockUpDown.commands.reset := #_w1 AND "Unit1.Em5.ControlNodes".cmCathodeNgBoxLockUpDown.monitoring.error;
   "Unit1.Em5.ControlNodes".cmCathodeNgPnpVaccum.commands.reset := #_w1 AND "Unit1.Em5.ControlNodes".cmCathodeNgPnpVaccum.monitoring.error;
   "Unit1.Em5.ControlNodes".cmCathodeConveyorCoverFwdBwd.commands.reset := #_w1 AND "Unit1.Em5.ControlNodes".cmCathodeConveyorCoverFwdBwd.monitoring.error;
   "Unit1.Em5.ControlNodes".cmCathodeConveyorPickUpBlower.commands.reset := #_w1 AND "Unit1.Em5.ControlNodes".cmCathodeConveyorPickUpBlower.monitoring.error;
END_REGION

REGION Network 223: CmCathodeMainPnP1RotaryCwCcw Home
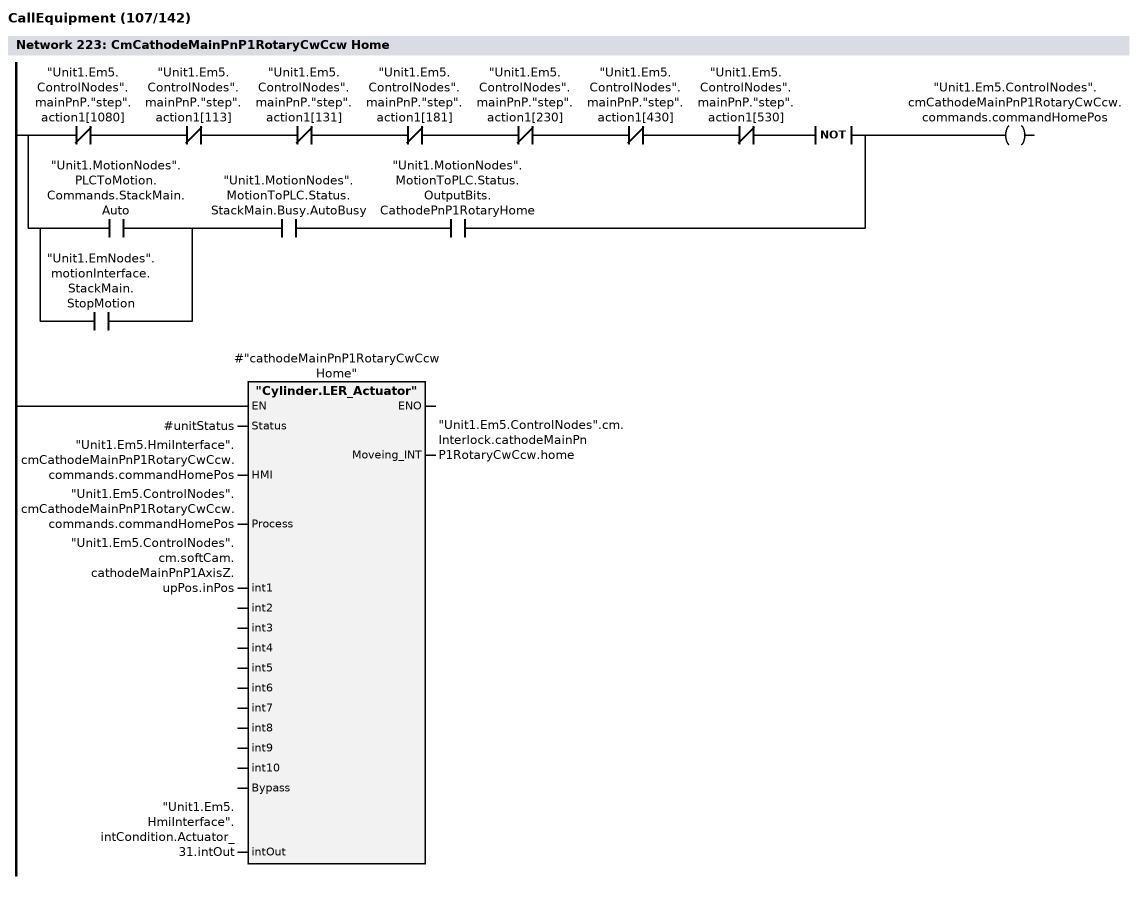
   RUNG wire#powerrail
      I_Contact( "Unit1.Em5.ControlNodes".mainPnP."step".action1[1080] )
      I_Contact( "Unit1.Em5.ControlNodes".mainPnP."step".action1[113] )
      I_Contact( "Unit1.Em5.ControlNodes".mainPnP."step".action1[131] )
      I_Contact( "Unit1.Em5.ControlNodes".mainPnP."step".action1[181] )
      I_Contact( "Unit1.Em5.ControlNodes".mainPnP."step".action1[230] )
      I_Contact( "Unit1.Em5.ControlNodes".mainPnP."step".action1[430] )
      I_Contact( "Unit1.Em5.ControlNodes".mainPnP."step".action1[530] )
      Not()
      wire#w1
      Coil( "Unit1.Em5.ControlNodes".cmCathodeMainPnP1RotaryCwCcw.commands.commandHomePos )
   END_RUNG
   RUNG wire#powerrail
      Contact( "Unit1.MotionNodes".PLCToMotion.Commands.StackMain.Auto )
      wire#w2
      Contact( "Unit1.MotionNodes".MotionToPLC.Status.StackMain.Busy.AutoBusy )
      Contact( "Unit1.MotionNodes".MotionToPLC.Status.OutputBits.CathodePnP1RotaryHome )
   END_RUNG wire#w1
   RUNG wire#powerrail
      Contact( "Unit1.EmNodes".motionInterface.StackMain.StopMotion )
   END_RUNG wire#w2
   RUNG wire#powerrail
      #"cathodeMainPnP1RotaryCwCcw Home"(Status := #unitStatus, HMI := "Unit1.Em5.HmiInterface".cmCathodeMainPnP1RotaryCwCcw.commands.commandHomePos, Process := "Unit1.Em5.ControlNodes".cmCathodeMainPnP1RotaryCwCcw.commands.commandHomePos, int1 := "Unit1.Em5.ControlNodes".cm.softCam.cathodeMainPnP1AxisZ.upPos.inPos, int2 :=, int3 :=, int4 :=, int5 :=, int6 :=, int7 :=, int8 :=, int9 :=, int10 :=, Bypass :=, intOut := "Unit1.Em5.HmiInterface".intCondition.Actuator_31.intOut, Moveing_INT => "Unit1.Em5.ControlNodes".cm.Interlock.cathodeMainPnP1RotaryCwCcw.home)
   END_RUNG
   // the same network as SCL:
   "Unit1.Em5.ControlNodes".cmCathodeMainPnP1RotaryCwCcw.commands.commandHomePos := NOT (NOT "Unit1.Em5.ControlNodes".mainPnP."step".action1[1080] AND NOT "Unit1.Em5.ControlNodes".mainPnP."step".action1[113] AND NOT "Unit1.Em5.ControlNodes".mainPnP."step".action1[131] AND NOT "Unit1.Em5.ControlNodes".mainPnP."step".action1[181] AND NOT "Unit1.Em5.ControlNodes".mainPnP."step".action1[230] AND NOT "Unit1.Em5.ControlNodes".mainPnP."step".action1[430] AND NOT "Unit1.Em5.ControlNodes".mainPnP."step".action1[530]) OR (("Unit1.MotionNodes".PLCToMotion.Commands.StackMain.Auto OR "Unit1.EmNodes".motionInterface.StackMain.StopMotion) AND "Unit1.MotionNodes".MotionToPLC.Status.StackMain.Busy.AutoBusy AND "Unit1.MotionNodes".MotionToPLC.Status.OutputBits.CathodePnP1RotaryHome);
   #"cathodeMainPnP1RotaryCwCcw Home"(Status := #unitStatus,   // "Cylinder.LER_Actuator"
                           HMI := "Unit1.Em5.HmiInterface".cmCathodeMainPnP1RotaryCwCcw.commands.commandHomePos,
                           Process := "Unit1.Em5.ControlNodes".cmCathodeMainPnP1RotaryCwCcw.commands.commandHomePos,
                           int1 := "Unit1.Em5.ControlNodes".cm.softCam.cathodeMainPnP1AxisZ.upPos.inPos,
                           intOut := "Unit1.Em5.HmiInterface".intCondition.Actuator_31.intOut,
                           Moveing_INT => "Unit1.Em5.ControlNodes".cm.Interlock.cathodeMainPnP1RotaryCwCcw.home);
END_REGION

REGION Network 224: CmCathodeMainPnP1RotaryCwCcw Work
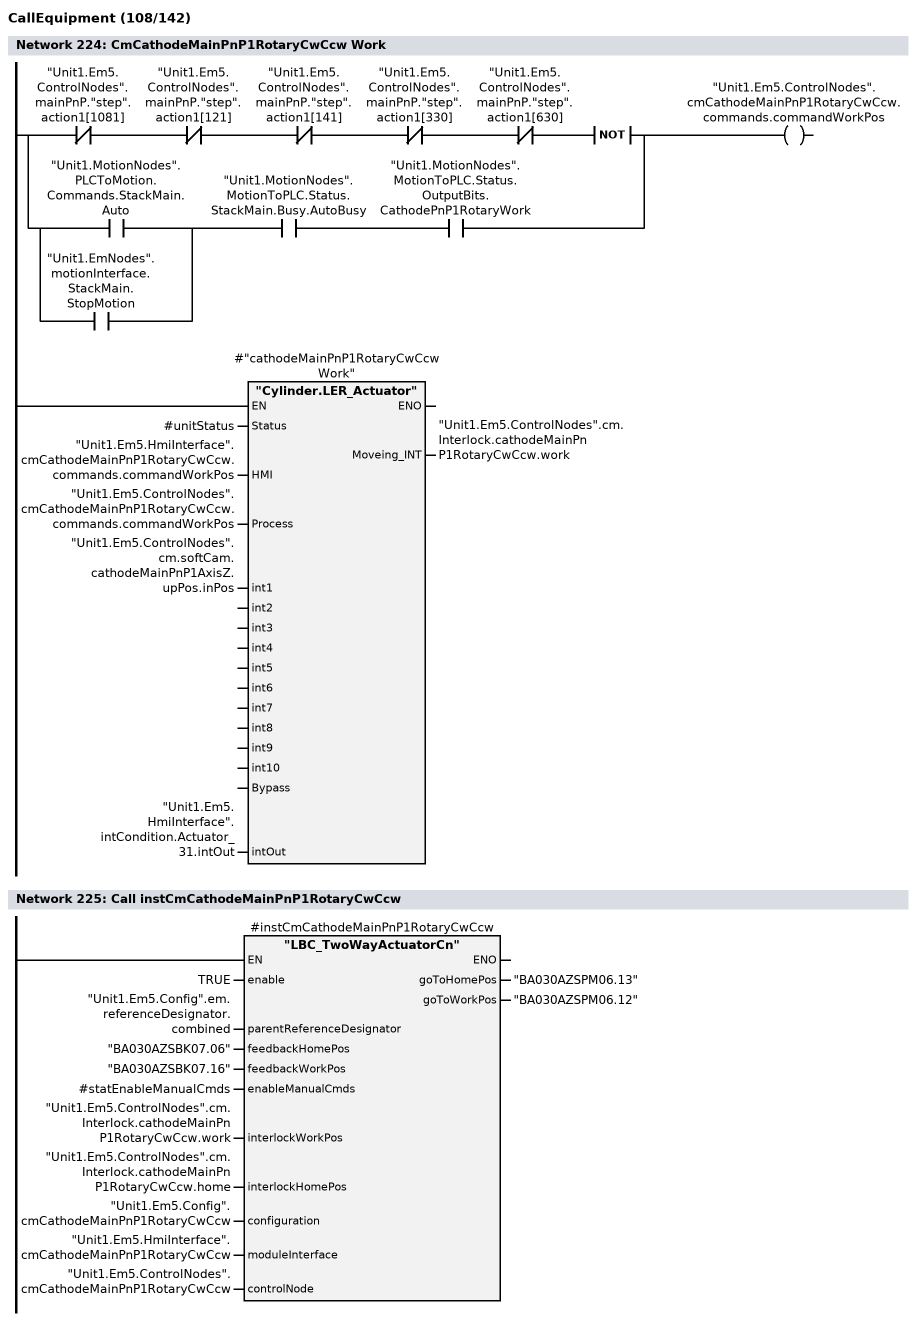
   RUNG wire#powerrail
      I_Contact( "Unit1.Em5.ControlNodes".mainPnP."step".action1[1081] )
      I_Contact( "Unit1.Em5.ControlNodes".mainPnP."step".action1[121] )
      I_Contact( "Unit1.Em5.ControlNodes".mainPnP."step".action1[141] )
      I_Contact( "Unit1.Em5.ControlNodes".mainPnP."step".action1[330] )
      I_Contact( "Unit1.Em5.ControlNodes".mainPnP."step".action1[630] )
      Not()
      wire#w1
      Coil( "Unit1.Em5.ControlNodes".cmCathodeMainPnP1RotaryCwCcw.commands.commandWorkPos )
   END_RUNG
   RUNG wire#powerrail
      Contact( "Unit1.MotionNodes".PLCToMotion.Commands.StackMain.Auto )
      wire#w2
      Contact( "Unit1.MotionNodes".MotionToPLC.Status.StackMain.Busy.AutoBusy )
      Contact( "Unit1.MotionNodes".MotionToPLC.Status.OutputBits.CathodePnP1RotaryWork )
   END_RUNG wire#w1
   RUNG wire#powerrail
      Contact( "Unit1.EmNodes".motionInterface.StackMain.StopMotion )
   END_RUNG wire#w2
   RUNG wire#powerrail
      #"cathodeMainPnP1RotaryCwCcw Work"(Status := #unitStatus, HMI := "Unit1.Em5.HmiInterface".cmCathodeMainPnP1RotaryCwCcw.commands.commandWorkPos, Process := "Unit1.Em5.ControlNodes".cmCathodeMainPnP1RotaryCwCcw.commands.commandWorkPos, int1 := "Unit1.Em5.ControlNodes".cm.softCam.cathodeMainPnP1AxisZ.upPos.inPos, int2 :=, int3 :=, int4 :=, int5 :=, int6 :=, int7 :=, int8 :=, int9 :=, int10 :=, Bypass :=, intOut := "Unit1.Em5.HmiInterface".intCondition.Actuator_31.intOut, Moveing_INT => "Unit1.Em5.ControlNodes".cm.Interlock.cathodeMainPnP1RotaryCwCcw.work)
   END_RUNG
   // the same network as SCL:
   "Unit1.Em5.ControlNodes".cmCathodeMainPnP1RotaryCwCcw.commands.commandWorkPos := NOT (NOT "Unit1.Em5.ControlNodes".mainPnP."step".action1[1081] AND NOT "Unit1.Em5.ControlNodes".mainPnP."step".action1[121] AND NOT "Unit1.Em5.ControlNodes".mainPnP."step".action1[141] AND NOT "Unit1.Em5.ControlNodes".mainPnP."step".action1[330] AND NOT "Unit1.Em5.ControlNodes".mainPnP."step".action1[630]) OR (("Unit1.MotionNodes".PLCToMotion.Commands.StackMain.Auto OR "Unit1.EmNodes".motionInterface.StackMain.StopMotion) AND "Unit1.MotionNodes".MotionToPLC.Status.StackMain.Busy.AutoBusy AND "Unit1.MotionNodes".MotionToPLC.Status.OutputBits.CathodePnP1RotaryWork);
   #"cathodeMainPnP1RotaryCwCcw Work"(Status := #unitStatus,   // "Cylinder.LER_Actuator"
                           HMI := "Unit1.Em5.HmiInterface".cmCathodeMainPnP1RotaryCwCcw.commands.commandWorkPos,
                           Process := "Unit1.Em5.ControlNodes".cmCathodeMainPnP1RotaryCwCcw.commands.commandWorkPos,
                           int1 := "Unit1.Em5.ControlNodes".cm.softCam.cathodeMainPnP1AxisZ.upPos.inPos,
                           intOut := "Unit1.Em5.HmiInterface".intCondition.Actuator_31.intOut,
                           Moveing_INT => "Unit1.Em5.ControlNodes".cm.Interlock.cathodeMainPnP1RotaryCwCcw.work);
END_REGION

REGION Network 225: Call instCmCathodeMainPnP1RotaryCwCcw
   RUNG wire#powerrail
      #instCmCathodeMainPnP1RotaryCwCcw(enable := TRUE, parentReferenceDesignator := "Unit1.Em5.Config".em.referenceDesignator.combined, feedbackHomePos := "BA030AZSBK07.06", feedbackWorkPos := "BA030AZSBK07.16", enableManualCmds := #statEnableManualCmds, interlockWorkPos := "Unit1.Em5.ControlNodes".cm.Interlock.cathodeMainPnP1RotaryCwCcw.work, interlockHomePos := "Unit1.Em5.ControlNodes".cm.Interlock.cathodeMainPnP1RotaryCwCcw.home, configuration := "Unit1.Em5.Config".cmCathodeMainPnP1RotaryCwCcw, moduleInterface := "Unit1.Em5.HmiInterface".cmCathodeMainPnP1RotaryCwCcw, controlNode := "Unit1.Em5.ControlNodes".cmCathodeMainPnP1RotaryCwCcw, goToHomePos => "BA030AZSPM06.13", goToWorkPos => "BA030AZSPM06.12")
   END_RUNG
   // the same network as SCL:
   #instCmCathodeMainPnP1RotaryCwCcw(enable := TRUE,   // "LBC_TwoWayActuatorCn"
                           parentReferenceDesignator := "Unit1.Em5.Config".em.referenceDesignator.combined,
                           feedbackHomePos := "BA030AZSBK07.06",
                           feedbackWorkPos := "BA030AZSBK07.16",
                           enableManualCmds := #statEnableManualCmds,
                           interlockWorkPos := "Unit1.Em5.ControlNodes".cm.Interlock.cathodeMainPnP1RotaryCwCcw.work,
                           interlockHomePos := "Unit1.Em5.ControlNodes".cm.Interlock.cathodeMainPnP1RotaryCwCcw.home,
                           configuration := "Unit1.Em5.Config".cmCathodeMainPnP1RotaryCwCcw,
                           moduleInterface := "Unit1.Em5.HmiInterface".cmCathodeMainPnP1RotaryCwCcw,
                           controlNode := "Unit1.Em5.ControlNodes".cmCathodeMainPnP1RotaryCwCcw,
                           goToHomePos => "BA030AZSPM06.13",
                           goToWorkPos => "BA030AZSPM06.12");
END_REGION

REGION Network 227: CmCathodeMainPnP1SuctionPlateVacuum Home
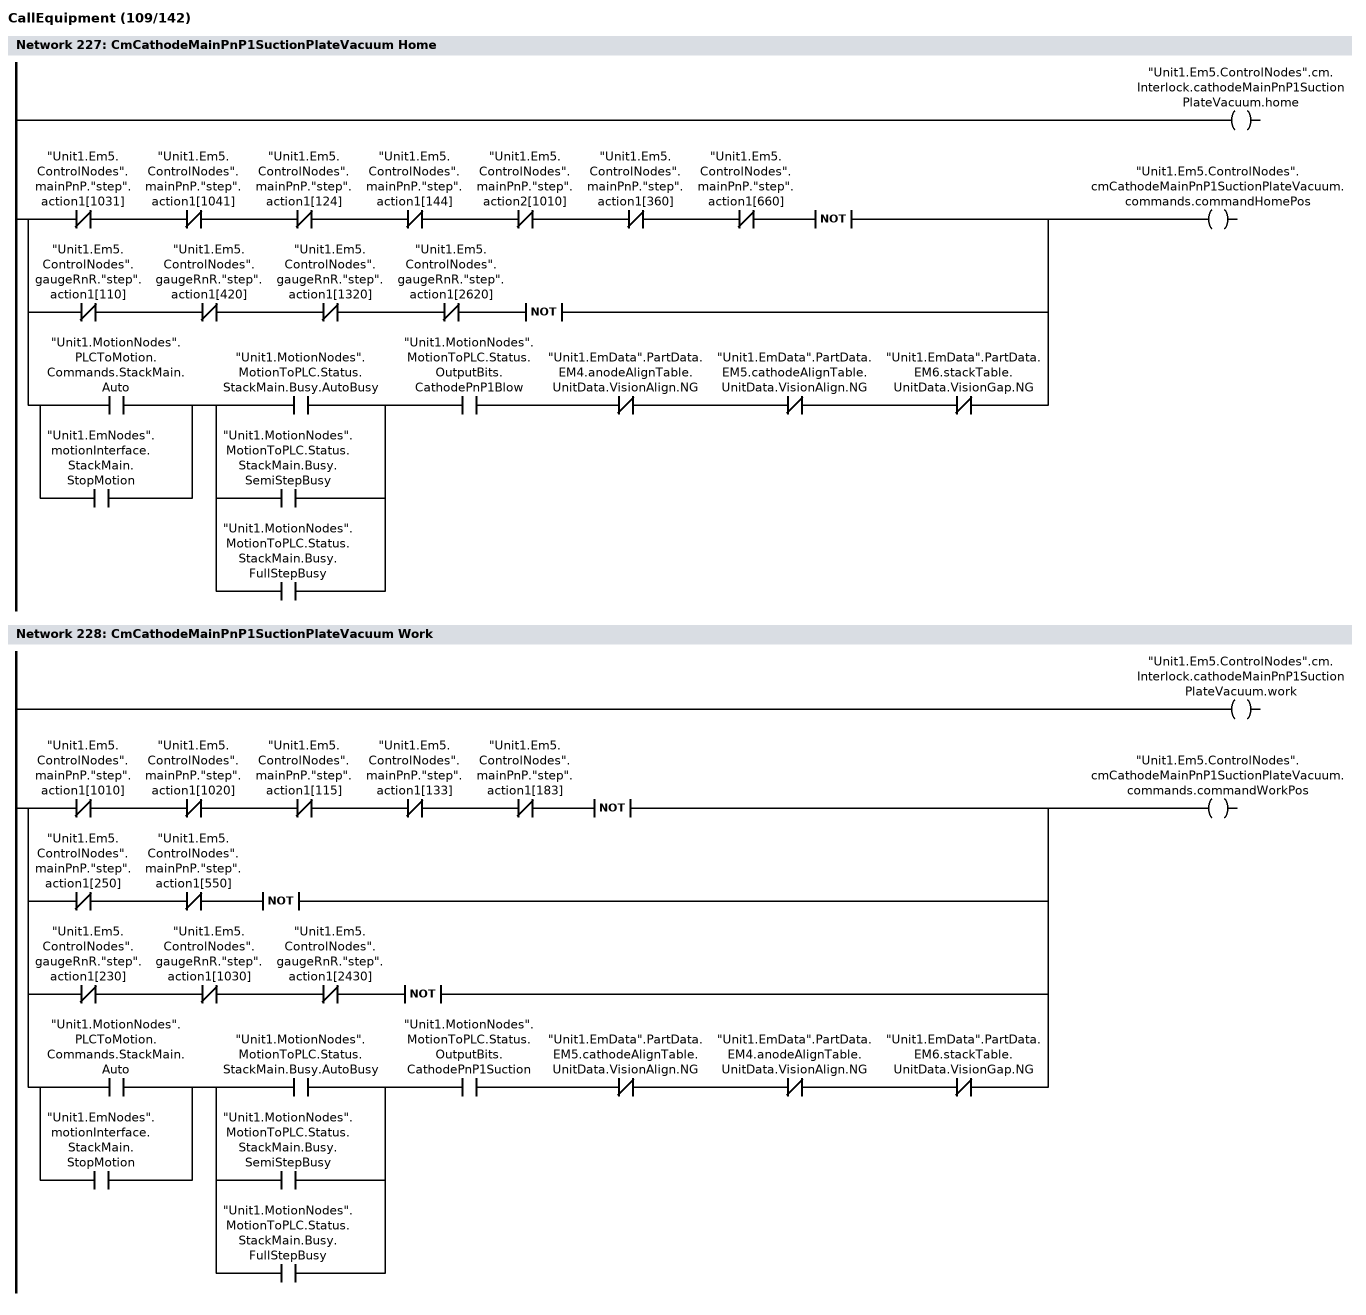
   RUNG wire#powerrail
      Coil( "Unit1.Em5.ControlNodes".cm.Interlock.cathodeMainPnP1SuctionPlateVacuum.home )
   END_RUNG
   RUNG wire#powerrail
      I_Contact( "Unit1.Em5.ControlNodes".mainPnP."step".action1[1031] )
      I_Contact( "Unit1.Em5.ControlNodes".mainPnP."step".action1[1041] )
      I_Contact( "Unit1.Em5.ControlNodes".mainPnP."step".action1[124] )
      I_Contact( "Unit1.Em5.ControlNodes".mainPnP."step".action1[144] )
      I_Contact( "Unit1.Em5.ControlNodes".mainPnP."step".action2[1010] )
      I_Contact( "Unit1.Em5.ControlNodes".mainPnP."step".action1[360] )
      I_Contact( "Unit1.Em5.ControlNodes".mainPnP."step".action1[660] )
      Not()
      wire#w1
      Coil( "Unit1.Em5.ControlNodes".cmCathodeMainPnP1SuctionPlateVacuum.commands.commandHomePos )
   END_RUNG
   RUNG wire#powerrail
      I_Contact( "Unit1.Em5.ControlNodes".gaugeRnR."step".action1[110] )
      I_Contact( "Unit1.Em5.ControlNodes".gaugeRnR."step".action1[420] )
      I_Contact( "Unit1.Em5.ControlNodes".gaugeRnR."step".action1[1320] )
      I_Contact( "Unit1.Em5.ControlNodes".gaugeRnR."step".action1[2620] )
      Not()
   END_RUNG wire#w1
   RUNG wire#powerrail
      Contact( "Unit1.MotionNodes".PLCToMotion.Commands.StackMain.Auto )
      wire#w2
      Contact( "Unit1.MotionNodes".MotionToPLC.Status.StackMain.Busy.AutoBusy )
      wire#w3
      Contact( "Unit1.MotionNodes".MotionToPLC.Status.OutputBits.CathodePnP1Blow )
      I_Contact( "Unit1.EmData".PartData.EM4.anodeAlignTable.UnitData.VisionAlign.NG )
      I_Contact( "Unit1.EmData".PartData.EM5.cathodeAlignTable.UnitData.VisionAlign.NG )
      I_Contact( "Unit1.EmData".PartData.EM6.stackTable.UnitData.VisionGap.NG )
   END_RUNG wire#w1
   RUNG wire#powerrail
      Contact( "Unit1.EmNodes".motionInterface.StackMain.StopMotion )
   END_RUNG wire#w2
   RUNG wire#w2
      Contact( "Unit1.MotionNodes".MotionToPLC.Status.StackMain.Busy.SemiStepBusy )
   END_RUNG wire#w3
   RUNG wire#w2
      Contact( "Unit1.MotionNodes".MotionToPLC.Status.StackMain.Busy.FullStepBusy )
   END_RUNG wire#w3
   // the same network as SCL:
   "Unit1.Em5.ControlNodes".cm.Interlock.cathodeMainPnP1SuctionPlateVacuum.home := TRUE;
   "Unit1.Em5.ControlNodes".cmCathodeMainPnP1SuctionPlateVacuum.commands.commandHomePos := NOT (NOT "Unit1.Em5.ControlNodes".mainPnP."step".action1[1031] AND NOT "Unit1.Em5.ControlNodes".mainPnP."step".action1[1041] AND NOT "Unit1.Em5.ControlNodes".mainPnP."step".action1[124] AND NOT "Unit1.Em5.ControlNodes".mainPnP."step".action1[144] AND NOT "Unit1.Em5.ControlNodes".mainPnP."step".action2[1010] AND NOT "Unit1.Em5.ControlNodes".mainPnP."step".action1[360] AND NOT "Unit1.Em5.ControlNodes".mainPnP."step".action1[660]) OR NOT (NOT "Unit1.Em5.ControlNodes".gaugeRnR."step".action1[110] AND NOT "Unit1.Em5.ControlNodes".gaugeRnR."step".action1[420] AND NOT "Unit1.Em5.ControlNodes".gaugeRnR."step".action1[1320] AND NOT "Unit1.Em5.ControlNodes".gaugeRnR."step".action1[2620]) OR (("Unit1.MotionNodes".PLCToMotion.Commands.StackMain.Auto OR "Unit1.EmNodes".motionInterface.StackMain.StopMotion) AND ("Unit1.MotionNodes".MotionToPLC.Status.StackMain.Busy.AutoBusy OR "Unit1.MotionNodes".MotionToPLC.Status.StackMain.Busy.SemiStepBusy OR "Unit1.MotionNodes".MotionToPLC.Status.StackMain.Busy.FullStepBusy) AND "Unit1.MotionNodes".MotionToPLC.Status.OutputBits.CathodePnP1Blow AND NOT "Unit1.EmData".PartData.EM4.anodeAlignTable.UnitData.VisionAlign.NG AND NOT "Unit1.EmData".PartData.EM5.cathodeAlignTable.UnitData.VisionAlign.NG AND NOT "Unit1.EmData".PartData.EM6.stackTable.UnitData.VisionGap.NG);
END_REGION

REGION Network 228: CmCathodeMainPnP1SuctionPlateVacuum Work
   RUNG wire#powerrail
      Coil( "Unit1.Em5.ControlNodes".cm.Interlock.cathodeMainPnP1SuctionPlateVacuum.work )
   END_RUNG
   RUNG wire#powerrail
      I_Contact( "Unit1.Em5.ControlNodes".mainPnP."step".action1[1010] )
      I_Contact( "Unit1.Em5.ControlNodes".mainPnP."step".action1[1020] )
      I_Contact( "Unit1.Em5.ControlNodes".mainPnP."step".action1[115] )
      I_Contact( "Unit1.Em5.ControlNodes".mainPnP."step".action1[133] )
      I_Contact( "Unit1.Em5.ControlNodes".mainPnP."step".action1[183] )
      Not()
      wire#w1
      Coil( "Unit1.Em5.ControlNodes".cmCathodeMainPnP1SuctionPlateVacuum.commands.commandWorkPos )
   END_RUNG
   RUNG wire#powerrail
      I_Contact( "Unit1.Em5.ControlNodes".mainPnP."step".action1[250] )
      I_Contact( "Unit1.Em5.ControlNodes".mainPnP."step".action1[550] )
      Not()
   END_RUNG wire#w1
   RUNG wire#powerrail
      I_Contact( "Unit1.Em5.ControlNodes".gaugeRnR."step".action1[230] )
      I_Contact( "Unit1.Em5.ControlNodes".gaugeRnR."step".action1[1030] )
      I_Contact( "Unit1.Em5.ControlNodes".gaugeRnR."step".action1[2430] )
      Not()
   END_RUNG wire#w1
   RUNG wire#powerrail
      Contact( "Unit1.MotionNodes".PLCToMotion.Commands.StackMain.Auto )
      wire#w2
      Contact( "Unit1.MotionNodes".MotionToPLC.Status.StackMain.Busy.AutoBusy )
      wire#w3
      Contact( "Unit1.MotionNodes".MotionToPLC.Status.OutputBits.CathodePnP1Suction )
      I_Contact( "Unit1.EmData".PartData.EM5.cathodeAlignTable.UnitData.VisionAlign.NG )
      I_Contact( "Unit1.EmData".PartData.EM4.anodeAlignTable.UnitData.VisionAlign.NG )
      I_Contact( "Unit1.EmData".PartData.EM6.stackTable.UnitData.VisionGap.NG )
   END_RUNG wire#w1
   RUNG wire#powerrail
      Contact( "Unit1.EmNodes".motionInterface.StackMain.StopMotion )
   END_RUNG wire#w2
   RUNG wire#w2
      Contact( "Unit1.MotionNodes".MotionToPLC.Status.StackMain.Busy.SemiStepBusy )
   END_RUNG wire#w3
   RUNG wire#w2
      Contact( "Unit1.MotionNodes".MotionToPLC.Status.StackMain.Busy.FullStepBusy )
   END_RUNG wire#w3
   // the same network as SCL:
   "Unit1.Em5.ControlNodes".cm.Interlock.cathodeMainPnP1SuctionPlateVacuum.work := TRUE;
   "Unit1.Em5.ControlNodes".cmCathodeMainPnP1SuctionPlateVacuum.commands.commandWorkPos := NOT (NOT "Unit1.Em5.ControlNodes".mainPnP."step".action1[1010] AND NOT "Unit1.Em5.ControlNodes".mainPnP."step".action1[1020] AND NOT "Unit1.Em5.ControlNodes".mainPnP."step".action1[115] AND NOT "Unit1.Em5.ControlNodes".mainPnP."step".action1[133] AND NOT "Unit1.Em5.ControlNodes".mainPnP."step".action1[183]) OR NOT (NOT "Unit1.Em5.ControlNodes".mainPnP."step".action1[250] AND NOT "Unit1.Em5.ControlNodes".mainPnP."step".action1[550]) OR NOT (NOT "Unit1.Em5.ControlNodes".gaugeRnR."step".action1[230] AND NOT "Unit1.Em5.ControlNodes".gaugeRnR."step".action1[1030] AND NOT "Unit1.Em5.ControlNodes".gaugeRnR."step".action1[2430]) OR (("Unit1.MotionNodes".PLCToMotion.Commands.StackMain.Auto OR "Unit1.EmNodes".motionInterface.StackMain.StopMotion) AND ("Unit1.MotionNodes".MotionToPLC.Status.StackMain.Busy.AutoBusy OR "Unit1.MotionNodes".MotionToPLC.Status.StackMain.Busy.SemiStepBusy OR "Unit1.MotionNodes".MotionToPLC.Status.StackMain.Busy.FullStepBusy) AND "Unit1.MotionNodes".MotionToPLC.Status.OutputBits.CathodePnP1Suction AND NOT "Unit1.EmData".PartData.EM5.cathodeAlignTable.UnitData.VisionAlign.NG AND NOT "Unit1.EmData".PartData.EM4.anodeAlignTable.UnitData.VisionAlign.NG AND NOT "Unit1.EmData".PartData.EM6.stackTable.UnitData.VisionGap.NG);
END_REGION

REGION Network 229: Call instCmCathodeMainPnP1SuctionPlateVacuum
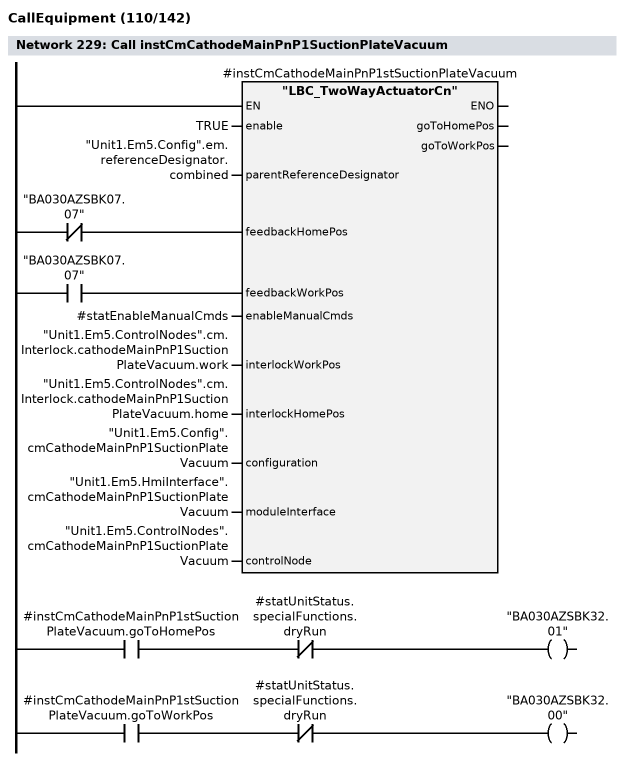
   RUNG wire#powerrail
      #instCmCathodeMainPnP1stSuctionPlateVacuum(feedbackHomePos := wire#w1, feedbackWorkPos := wire#w2, enable := TRUE, parentReferenceDesignator := "Unit1.Em5.Config".em.referenceDesignator.combined, enableManualCmds := #statEnableManualCmds, interlockWorkPos := "Unit1.Em5.ControlNodes".cm.Interlock.cathodeMainPnP1SuctionPlateVacuum.work, interlockHomePos := "Unit1.Em5.ControlNodes".cm.Interlock.cathodeMainPnP1SuctionPlateVacuum.home, configuration := "Unit1.Em5.Config".cmCathodeMainPnP1SuctionPlateVacuum, moduleInterface := "Unit1.Em5.HmiInterface".cmCathodeMainPnP1SuctionPlateVacuum, controlNode := "Unit1.Em5.ControlNodes".cmCathodeMainPnP1SuctionPlateVacuum, goToHomePos =>, goToWorkPos =>)
   END_RUNG
   RUNG wire#powerrail
      I_Contact( "BA030AZSBK07.07" )
   END_RUNG wire#w1
   RUNG wire#powerrail
      Contact( "BA030AZSBK07.07" )
   END_RUNG wire#w2
   RUNG wire#powerrail
      Contact( #instCmCathodeMainPnP1stSuctionPlateVacuum.goToHomePos )
      I_Contact( #statUnitStatus.specialFunctions.dryRun )
      Coil( "BA030AZSBK32.01" )
   END_RUNG
   RUNG wire#powerrail
      Contact( #instCmCathodeMainPnP1stSuctionPlateVacuum.goToWorkPos )
      I_Contact( #statUnitStatus.specialFunctions.dryRun )
      Coil( "BA030AZSBK32.00" )
   END_RUNG
   // the same network as SCL:
   #instCmCathodeMainPnP1stSuctionPlateVacuum(enable := TRUE,   // "LBC_TwoWayActuatorCn"
                           parentReferenceDesignator := "Unit1.Em5.Config".em.referenceDesignator.combined,
                           feedbackHomePos := NOT "BA030AZSBK07.07",
                           feedbackWorkPos := "BA030AZSBK07.07",
                           enableManualCmds := #statEnableManualCmds,
                           interlockWorkPos := "Unit1.Em5.ControlNodes".cm.Interlock.cathodeMainPnP1SuctionPlateVacuum.work,
                           interlockHomePos := "Unit1.Em5.ControlNodes".cm.Interlock.cathodeMainPnP1SuctionPlateVacuum.home,
                           configuration := "Unit1.Em5.Config".cmCathodeMainPnP1SuctionPlateVacuum,
                           moduleInterface := "Unit1.Em5.HmiInterface".cmCathodeMainPnP1SuctionPlateVacuum,
                           controlNode := "Unit1.Em5.ControlNodes".cmCathodeMainPnP1SuctionPlateVacuum);
   "BA030AZSBK32.01" := #instCmCathodeMainPnP1stSuctionPlateVacuum.goToHomePos AND NOT #statUnitStatus.specialFunctions.dryRun;
   "BA030AZSBK32.00" := #instCmCathodeMainPnP1stSuctionPlateVacuum.goToWorkPos AND NOT #statUnitStatus.specialFunctions.dryRun;
END_REGION

REGION Network 231: CmCathodeMainPnP2SuctionPlateVacuum Home
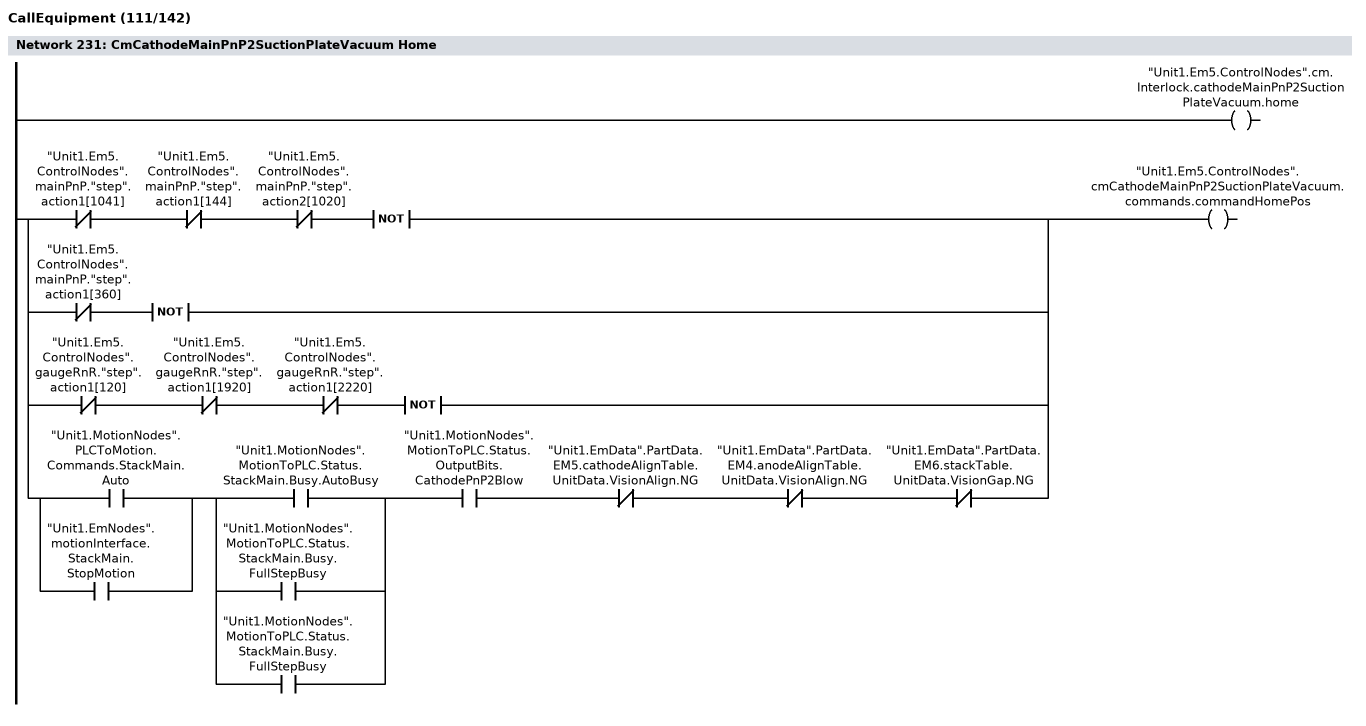
   RUNG wire#powerrail
      Coil( "Unit1.Em5.ControlNodes".cm.Interlock.cathodeMainPnP2SuctionPlateVacuum.home )
   END_RUNG
   RUNG wire#powerrail
      I_Contact( "Unit1.Em5.ControlNodes".mainPnP."step".action1[1041] )
      I_Contact( "Unit1.Em5.ControlNodes".mainPnP."step".action1[144] )
      I_Contact( "Unit1.Em5.ControlNodes".mainPnP."step".action2[1020] )
      Not()
      wire#w1
      Coil( "Unit1.Em5.ControlNodes".cmCathodeMainPnP2SuctionPlateVacuum.commands.commandHomePos )
   END_RUNG
   RUNG wire#powerrail
      I_Contact( "Unit1.Em5.ControlNodes".mainPnP."step".action1[360] )
      Not()
   END_RUNG wire#w1
   RUNG wire#powerrail
      I_Contact( "Unit1.Em5.ControlNodes".gaugeRnR."step".action1[120] )
      I_Contact( "Unit1.Em5.ControlNodes".gaugeRnR."step".action1[1920] )
      I_Contact( "Unit1.Em5.ControlNodes".gaugeRnR."step".action1[2220] )
      Not()
   END_RUNG wire#w1
   RUNG wire#powerrail
      Contact( "Unit1.MotionNodes".PLCToMotion.Commands.StackMain.Auto )
      wire#w2
      Contact( "Unit1.MotionNodes".MotionToPLC.Status.StackMain.Busy.AutoBusy )
      wire#w3
      Contact( "Unit1.MotionNodes".MotionToPLC.Status.OutputBits.CathodePnP2Blow )
      I_Contact( "Unit1.EmData".PartData.EM5.cathodeAlignTable.UnitData.VisionAlign.NG )
      I_Contact( "Unit1.EmData".PartData.EM4.anodeAlignTable.UnitData.VisionAlign.NG )
      I_Contact( "Unit1.EmData".PartData.EM6.stackTable.UnitData.VisionGap.NG )
   END_RUNG wire#w1
   RUNG wire#powerrail
      Contact( "Unit1.EmNodes".motionInterface.StackMain.StopMotion )
   END_RUNG wire#w2
   RUNG wire#w2
      Contact( "Unit1.MotionNodes".MotionToPLC.Status.StackMain.Busy.FullStepBusy )
   END_RUNG wire#w3
   RUNG wire#w2
      Contact( "Unit1.MotionNodes".MotionToPLC.Status.StackMain.Busy.FullStepBusy )
   END_RUNG wire#w3
   // the same network as SCL:
   "Unit1.Em5.ControlNodes".cm.Interlock.cathodeMainPnP2SuctionPlateVacuum.home := TRUE;
   "Unit1.Em5.ControlNodes".cmCathodeMainPnP2SuctionPlateVacuum.commands.commandHomePos := NOT (NOT "Unit1.Em5.ControlNodes".mainPnP."step".action1[1041] AND NOT "Unit1.Em5.ControlNodes".mainPnP."step".action1[144] AND NOT "Unit1.Em5.ControlNodes".mainPnP."step".action2[1020]) OR NOT (NOT "Unit1.Em5.ControlNodes".mainPnP."step".action1[360]) OR NOT (NOT "Unit1.Em5.ControlNodes".gaugeRnR."step".action1[120] AND NOT "Unit1.Em5.ControlNodes".gaugeRnR."step".action1[1920] AND NOT "Unit1.Em5.ControlNodes".gaugeRnR."step".action1[2220]) OR (("Unit1.MotionNodes".PLCToMotion.Commands.StackMain.Auto OR "Unit1.EmNodes".motionInterface.StackMain.StopMotion) AND ("Unit1.MotionNodes".MotionToPLC.Status.StackMain.Busy.AutoBusy OR "Unit1.MotionNodes".MotionToPLC.Status.StackMain.Busy.FullStepBusy OR "Unit1.MotionNodes".MotionToPLC.Status.StackMain.Busy.FullStepBusy) AND "Unit1.MotionNodes".MotionToPLC.Status.OutputBits.CathodePnP2Blow AND NOT "Unit1.EmData".PartData.EM5.cathodeAlignTable.UnitData.VisionAlign.NG AND NOT "Unit1.EmData".PartData.EM4.anodeAlignTable.UnitData.VisionAlign.NG AND NOT "Unit1.EmData".PartData.EM6.stackTable.UnitData.VisionGap.NG);
END_REGION

REGION Network 232: CmCathodeMainPnP2SuctionPlateVacuum Work
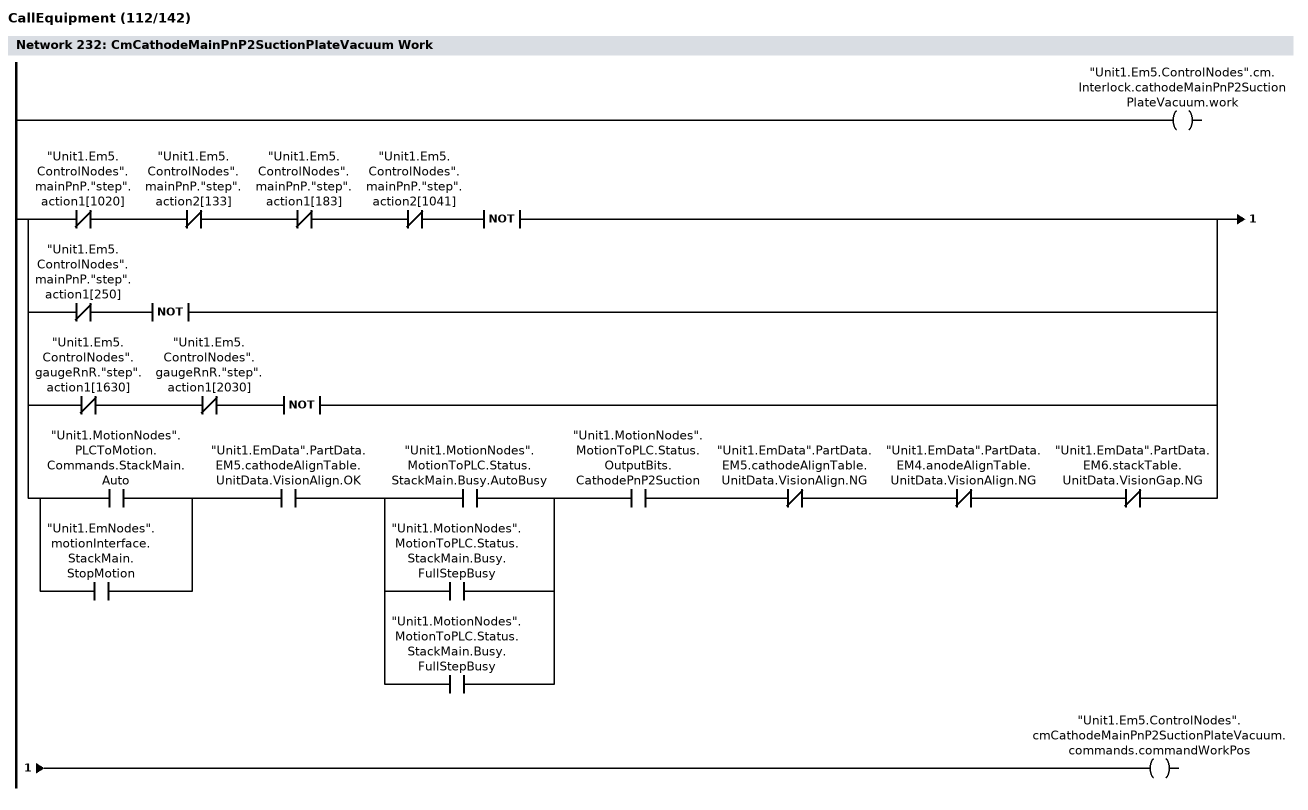
   RUNG wire#powerrail
      Coil( "Unit1.Em5.ControlNodes".cm.Interlock.cathodeMainPnP2SuctionPlateVacuum.work )
   END_RUNG
   RUNG wire#powerrail
      I_Contact( "Unit1.Em5.ControlNodes".mainPnP."step".action1[1020] )
      I_Contact( "Unit1.Em5.ControlNodes".mainPnP."step".action2[133] )
      I_Contact( "Unit1.Em5.ControlNodes".mainPnP."step".action1[183] )
      I_Contact( "Unit1.Em5.ControlNodes".mainPnP."step".action2[1041] )
      Not()
      wire#w1
      Coil( "Unit1.Em5.ControlNodes".cmCathodeMainPnP2SuctionPlateVacuum.commands.commandWorkPos )
   END_RUNG
   RUNG wire#powerrail
      I_Contact( "Unit1.Em5.ControlNodes".mainPnP."step".action1[250] )
      Not()
   END_RUNG wire#w1
   RUNG wire#powerrail
      I_Contact( "Unit1.Em5.ControlNodes".gaugeRnR."step".action1[1630] )
      I_Contact( "Unit1.Em5.ControlNodes".gaugeRnR."step".action1[2030] )
      Not()
   END_RUNG wire#w1
   RUNG wire#powerrail
      Contact( "Unit1.MotionNodes".PLCToMotion.Commands.StackMain.Auto )
      wire#w2
      Contact( "Unit1.EmData".PartData.EM5.cathodeAlignTable.UnitData.VisionAlign.OK )
      wire#w3
      Contact( "Unit1.MotionNodes".MotionToPLC.Status.StackMain.Busy.AutoBusy )
      wire#w4
      Contact( "Unit1.MotionNodes".MotionToPLC.Status.OutputBits.CathodePnP2Suction )
      I_Contact( "Unit1.EmData".PartData.EM5.cathodeAlignTable.UnitData.VisionAlign.NG )
      I_Contact( "Unit1.EmData".PartData.EM4.anodeAlignTable.UnitData.VisionAlign.NG )
      I_Contact( "Unit1.EmData".PartData.EM6.stackTable.UnitData.VisionGap.NG )
   END_RUNG wire#w1
   RUNG wire#powerrail
      Contact( "Unit1.EmNodes".motionInterface.StackMain.StopMotion )
   END_RUNG wire#w2
   RUNG wire#w3
      Contact( "Unit1.MotionNodes".MotionToPLC.Status.StackMain.Busy.FullStepBusy )
   END_RUNG wire#w4
   RUNG wire#w3
      Contact( "Unit1.MotionNodes".MotionToPLC.Status.StackMain.Busy.FullStepBusy )
   END_RUNG wire#w4
   // the same network as SCL:
   "Unit1.Em5.ControlNodes".cm.Interlock.cathodeMainPnP2SuctionPlateVacuum.work := TRUE;
   "Unit1.Em5.ControlNodes".cmCathodeMainPnP2SuctionPlateVacuum.commands.commandWorkPos := NOT (NOT "Unit1.Em5.ControlNodes".mainPnP."step".action1[1020] AND NOT "Unit1.Em5.ControlNodes".mainPnP."step".action2[133] AND NOT "Unit1.Em5.ControlNodes".mainPnP."step".action1[183] AND NOT "Unit1.Em5.ControlNodes".mainPnP."step".action2[1041]) OR NOT (NOT "Unit1.Em5.ControlNodes".mainPnP."step".action1[250]) OR NOT (NOT "Unit1.Em5.ControlNodes".gaugeRnR."step".action1[1630] AND NOT "Unit1.Em5.ControlNodes".gaugeRnR."step".action1[2030]) OR (("Unit1.MotionNodes".PLCToMotion.Commands.StackMain.Auto OR "Unit1.EmNodes".motionInterface.StackMain.StopMotion) AND "Unit1.EmData".PartData.EM5.cathodeAlignTable.UnitData.VisionAlign.OK AND ("Unit1.MotionNodes".MotionToPLC.Status.StackMain.Busy.AutoBusy OR "Unit1.MotionNodes".MotionToPLC.Status.StackMain.Busy.FullStepBusy OR "Unit1.MotionNodes".MotionToPLC.Status.StackMain.Busy.FullStepBusy) AND "Unit1.MotionNodes".MotionToPLC.Status.OutputBits.CathodePnP2Suction AND NOT "Unit1.EmData".PartData.EM5.cathodeAlignTable.UnitData.VisionAlign.NG AND NOT "Unit1.EmData".PartData.EM4.anodeAlignTable.UnitData.VisionAlign.NG AND NOT "Unit1.EmData".PartData.EM6.stackTable.UnitData.VisionGap.NG);
END_REGION

REGION Network 233: Call instCmCathodeMainPnP2SuctionPlateVacuum
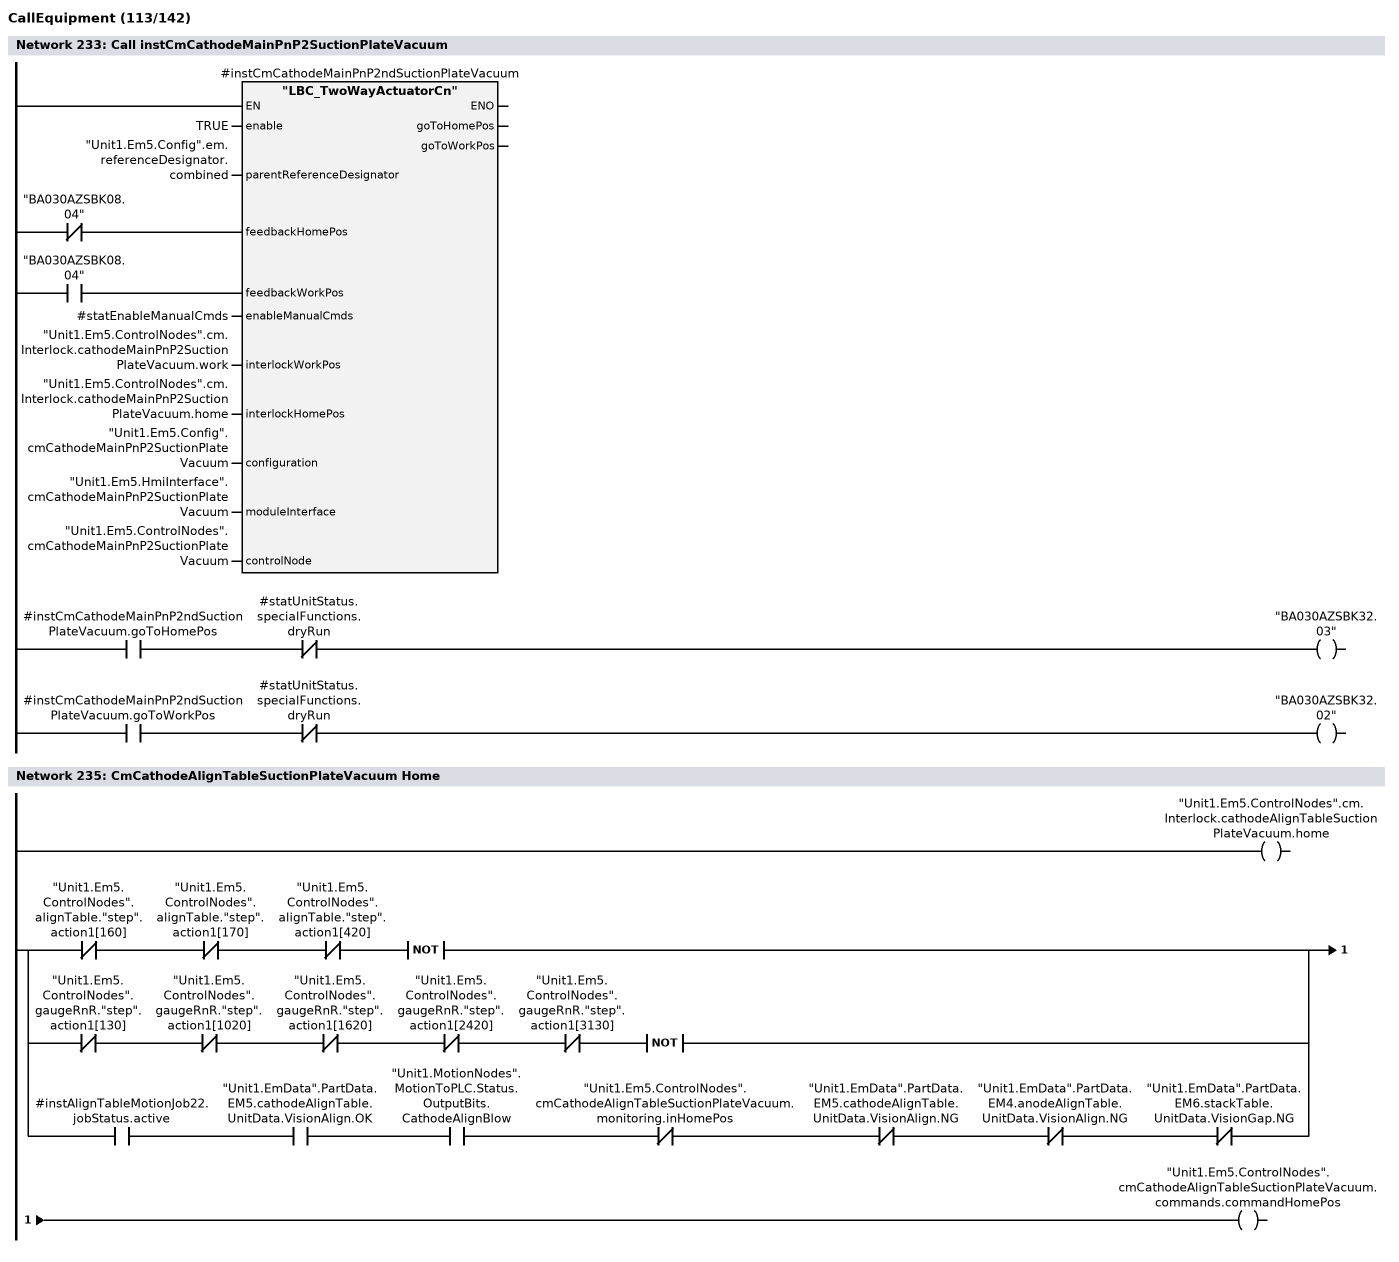
   RUNG wire#powerrail
      #instCmCathodeMainPnP2ndSuctionPlateVacuum(feedbackHomePos := wire#w1, feedbackWorkPos := wire#w2, enable := TRUE, parentReferenceDesignator := "Unit1.Em5.Config".em.referenceDesignator.combined, enableManualCmds := #statEnableManualCmds, interlockWorkPos := "Unit1.Em5.ControlNodes".cm.Interlock.cathodeMainPnP2SuctionPlateVacuum.work, interlockHomePos := "Unit1.Em5.ControlNodes".cm.Interlock.cathodeMainPnP2SuctionPlateVacuum.home, configuration := "Unit1.Em5.Config".cmCathodeMainPnP2SuctionPlateVacuum, moduleInterface := "Unit1.Em5.HmiInterface".cmCathodeMainPnP2SuctionPlateVacuum, controlNode := "Unit1.Em5.ControlNodes".cmCathodeMainPnP2SuctionPlateVacuum, goToHomePos =>, goToWorkPos =>)
   END_RUNG
   RUNG wire#powerrail
      I_Contact( "BA030AZSBK08.04" )
   END_RUNG wire#w1
   RUNG wire#powerrail
      Contact( "BA030AZSBK08.04" )
   END_RUNG wire#w2
   RUNG wire#powerrail
      Contact( #instCmCathodeMainPnP2ndSuctionPlateVacuum.goToHomePos )
      I_Contact( #statUnitStatus.specialFunctions.dryRun )
      Coil( "BA030AZSBK32.03" )
   END_RUNG
   RUNG wire#powerrail
      Contact( #instCmCathodeMainPnP2ndSuctionPlateVacuum.goToWorkPos )
      I_Contact( #statUnitStatus.specialFunctions.dryRun )
      Coil( "BA030AZSBK32.02" )
   END_RUNG
   // the same network as SCL:
   #instCmCathodeMainPnP2ndSuctionPlateVacuum(enable := TRUE,   // "LBC_TwoWayActuatorCn"
                           parentReferenceDesignator := "Unit1.Em5.Config".em.referenceDesignator.combined,
                           feedbackHomePos := NOT "BA030AZSBK08.04",
                           feedbackWorkPos := "BA030AZSBK08.04",
                           enableManualCmds := #statEnableManualCmds,
                           interlockWorkPos := "Unit1.Em5.ControlNodes".cm.Interlock.cathodeMainPnP2SuctionPlateVacuum.work,
                           interlockHomePos := "Unit1.Em5.ControlNodes".cm.Interlock.cathodeMainPnP2SuctionPlateVacuum.home,
                           configuration := "Unit1.Em5.Config".cmCathodeMainPnP2SuctionPlateVacuum,
                           moduleInterface := "Unit1.Em5.HmiInterface".cmCathodeMainPnP2SuctionPlateVacuum,
                           controlNode := "Unit1.Em5.ControlNodes".cmCathodeMainPnP2SuctionPlateVacuum);
   "BA030AZSBK32.03" := #instCmCathodeMainPnP2ndSuctionPlateVacuum.goToHomePos AND NOT #statUnitStatus.specialFunctions.dryRun;
   "BA030AZSBK32.02" := #instCmCathodeMainPnP2ndSuctionPlateVacuum.goToWorkPos AND NOT #statUnitStatus.specialFunctions.dryRun;
END_REGION

REGION Network 235: CmCathodeAlignTableSuctionPlateVacuum Home
   RUNG wire#powerrail
      Coil( "Unit1.Em5.ControlNodes".cm.Interlock.cathodeAlignTableSuctionPlateVacuum.home )
   END_RUNG
   RUNG wire#powerrail
      I_Contact( "Unit1.Em5.ControlNodes".alignTable."step".action1[160] )
      I_Contact( "Unit1.Em5.ControlNodes".alignTable."step".action1[170] )
      I_Contact( "Unit1.Em5.ControlNodes".alignTable."step".action1[420] )
      Not()
      wire#w1
      Coil( "Unit1.Em5.ControlNodes".cmCathodeAlignTableSuctionPlateVacuum.commands.commandHomePos )
   END_RUNG
   RUNG wire#powerrail
      I_Contact( "Unit1.Em5.ControlNodes".gaugeRnR."step".action1[130] )
      I_Contact( "Unit1.Em5.ControlNodes".gaugeRnR."step".action1[1020] )
      I_Contact( "Unit1.Em5.ControlNodes".gaugeRnR."step".action1[1620] )
      I_Contact( "Unit1.Em5.ControlNodes".gaugeRnR."step".action1[2420] )
      I_Contact( "Unit1.Em5.ControlNodes".gaugeRnR."step".action1[3130] )
      Not()
   END_RUNG wire#w1
   RUNG wire#powerrail
      Contact( #instAlignTableMotionJob22.jobStatus.active )
      Contact( "Unit1.EmData".PartData.EM5.cathodeAlignTable.UnitData.VisionAlign.OK )
      Contact( "Unit1.MotionNodes".MotionToPLC.Status.OutputBits.CathodeAlignBlow )
      I_Contact( "Unit1.Em5.ControlNodes".cmCathodeAlignTableSuctionPlateVacuum.monitoring.inHomePos )
      I_Contact( "Unit1.EmData".PartData.EM5.cathodeAlignTable.UnitData.VisionAlign.NG )
      I_Contact( "Unit1.EmData".PartData.EM4.anodeAlignTable.UnitData.VisionAlign.NG )
      I_Contact( "Unit1.EmData".PartData.EM6.stackTable.UnitData.VisionGap.NG )
   END_RUNG wire#w1
   // the same network as SCL:
   "Unit1.Em5.ControlNodes".cm.Interlock.cathodeAlignTableSuctionPlateVacuum.home := TRUE;
   "Unit1.Em5.ControlNodes".cmCathodeAlignTableSuctionPlateVacuum.commands.commandHomePos := NOT (NOT "Unit1.Em5.ControlNodes".alignTable."step".action1[160] AND NOT "Unit1.Em5.ControlNodes".alignTable."step".action1[170] AND NOT "Unit1.Em5.ControlNodes".alignTable."step".action1[420]) OR NOT (NOT "Unit1.Em5.ControlNodes".gaugeRnR."step".action1[130] AND NOT "Unit1.Em5.ControlNodes".gaugeRnR."step".action1[1020] AND NOT "Unit1.Em5.ControlNodes".gaugeRnR."step".action1[1620] AND NOT "Unit1.Em5.ControlNodes".gaugeRnR."step".action1[2420] AND NOT "Unit1.Em5.ControlNodes".gaugeRnR."step".action1[3130]) OR (#instAlignTableMotionJob22.jobStatus.active AND "Unit1.EmData".PartData.EM5.cathodeAlignTable.UnitData.VisionAlign.OK AND "Unit1.MotionNodes".MotionToPLC.Status.OutputBits.CathodeAlignBlow AND NOT "Unit1.Em5.ControlNodes".cmCathodeAlignTableSuctionPlateVacuum.monitoring.inHomePos AND NOT "Unit1.EmData".PartData.EM5.cathodeAlignTable.UnitData.VisionAlign.NG AND NOT "Unit1.EmData".PartData.EM4.anodeAlignTable.UnitData.VisionAlign.NG AND NOT "Unit1.EmData".PartData.EM6.stackTable.UnitData.VisionGap.NG);
END_REGION

REGION Network 236: CmCathodeAlginTableSuctionPlateVacuum Work
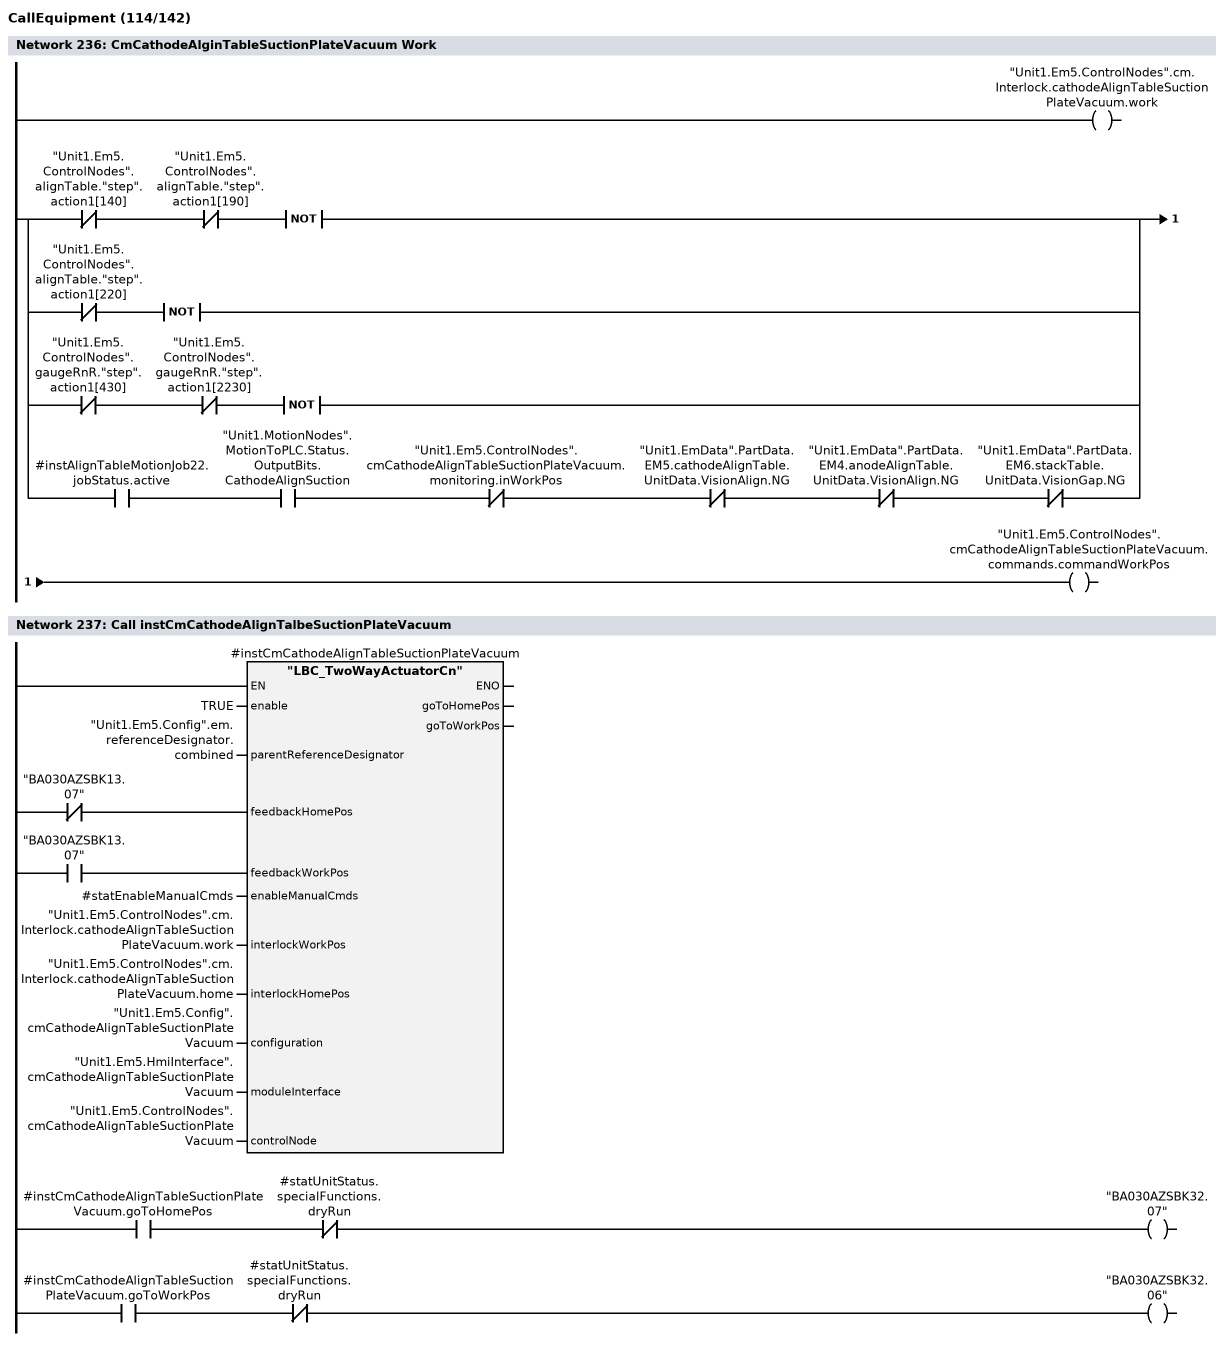
   RUNG wire#powerrail
      Coil( "Unit1.Em5.ControlNodes".cm.Interlock.cathodeAlignTableSuctionPlateVacuum.work )
   END_RUNG
   RUNG wire#powerrail
      I_Contact( "Unit1.Em5.ControlNodes".alignTable."step".action1[140] )
      I_Contact( "Unit1.Em5.ControlNodes".alignTable."step".action1[190] )
      Not()
      wire#w1
      Coil( "Unit1.Em5.ControlNodes".cmCathodeAlignTableSuctionPlateVacuum.commands.commandWorkPos )
   END_RUNG
   RUNG wire#powerrail
      I_Contact( "Unit1.Em5.ControlNodes".alignTable."step".action1[220] )
      Not()
   END_RUNG wire#w1
   RUNG wire#powerrail
      I_Contact( "Unit1.Em5.ControlNodes".gaugeRnR."step".action1[430] )
      I_Contact( "Unit1.Em5.ControlNodes".gaugeRnR."step".action1[2230] )
      Not()
   END_RUNG wire#w1
   RUNG wire#powerrail
      Contact( #instAlignTableMotionJob22.jobStatus.active )
      Contact( "Unit1.MotionNodes".MotionToPLC.Status.OutputBits.CathodeAlignSuction )
      I_Contact( "Unit1.Em5.ControlNodes".cmCathodeAlignTableSuctionPlateVacuum.monitoring.inWorkPos )
      I_Contact( "Unit1.EmData".PartData.EM5.cathodeAlignTable.UnitData.VisionAlign.NG )
      I_Contact( "Unit1.EmData".PartData.EM4.anodeAlignTable.UnitData.VisionAlign.NG )
      I_Contact( "Unit1.EmData".PartData.EM6.stackTable.UnitData.VisionGap.NG )
   END_RUNG wire#w1
   // the same network as SCL:
   "Unit1.Em5.ControlNodes".cm.Interlock.cathodeAlignTableSuctionPlateVacuum.work := TRUE;
   "Unit1.Em5.ControlNodes".cmCathodeAlignTableSuctionPlateVacuum.commands.commandWorkPos := NOT (NOT "Unit1.Em5.ControlNodes".alignTable."step".action1[140] AND NOT "Unit1.Em5.ControlNodes".alignTable."step".action1[190]) OR NOT (NOT "Unit1.Em5.ControlNodes".alignTable."step".action1[220]) OR NOT (NOT "Unit1.Em5.ControlNodes".gaugeRnR."step".action1[430] AND NOT "Unit1.Em5.ControlNodes".gaugeRnR."step".action1[2230]) OR (#instAlignTableMotionJob22.jobStatus.active AND "Unit1.MotionNodes".MotionToPLC.Status.OutputBits.CathodeAlignSuction AND NOT "Unit1.Em5.ControlNodes".cmCathodeAlignTableSuctionPlateVacuum.monitoring.inWorkPos AND NOT "Unit1.EmData".PartData.EM5.cathodeAlignTable.UnitData.VisionAlign.NG AND NOT "Unit1.EmData".PartData.EM4.anodeAlignTable.UnitData.VisionAlign.NG AND NOT "Unit1.EmData".PartData.EM6.stackTable.UnitData.VisionGap.NG);
END_REGION

REGION Network 237: Call instCmCathodeAlignTalbeSuctionPlateVacuum
   RUNG wire#powerrail
      #instCmCathodeAlignTableSuctionPlateVacuum(feedbackHomePos := wire#w1, feedbackWorkPos := wire#w2, enable := TRUE, parentReferenceDesignator := "Unit1.Em5.Config".em.referenceDesignator.combined, enableManualCmds := #statEnableManualCmds, interlockWorkPos := "Unit1.Em5.ControlNodes".cm.Interlock.cathodeAlignTableSuctionPlateVacuum.work, interlockHomePos := "Unit1.Em5.ControlNodes".cm.Interlock.cathodeAlignTableSuctionPlateVacuum.home, configuration := "Unit1.Em5.Config".cmCathodeAlignTableSuctionPlateVacuum, moduleInterface := "Unit1.Em5.HmiInterface".cmCathodeAlignTableSuctionPlateVacuum, controlNode := "Unit1.Em5.ControlNodes".cmCathodeAlignTableSuctionPlateVacuum, goToHomePos =>, goToWorkPos =>)
   END_RUNG
   RUNG wire#powerrail
      I_Contact( "BA030AZSBK13.07" )
   END_RUNG wire#w1
   RUNG wire#powerrail
      Contact( "BA030AZSBK13.07" )
   END_RUNG wire#w2
   RUNG wire#powerrail
      Contact( #instCmCathodeAlignTableSuctionPlateVacuum.goToHomePos )
      I_Contact( #statUnitStatus.specialFunctions.dryRun )
      Coil( "BA030AZSBK32.07" )
   END_RUNG
   RUNG wire#powerrail
      Contact( #instCmCathodeAlignTableSuctionPlateVacuum.goToWorkPos )
      I_Contact( #statUnitStatus.specialFunctions.dryRun )
      Coil( "BA030AZSBK32.06" )
   END_RUNG
   // the same network as SCL:
   #instCmCathodeAlignTableSuctionPlateVacuum(enable := TRUE,   // "LBC_TwoWayActuatorCn"
                           parentReferenceDesignator := "Unit1.Em5.Config".em.referenceDesignator.combined,
                           feedbackHomePos := NOT "BA030AZSBK13.07",
                           feedbackWorkPos := "BA030AZSBK13.07",
                           enableManualCmds := #statEnableManualCmds,
                           interlockWorkPos := "Unit1.Em5.ControlNodes".cm.Interlock.cathodeAlignTableSuctionPlateVacuum.work,
                           interlockHomePos := "Unit1.Em5.ControlNodes".cm.Interlock.cathodeAlignTableSuctionPlateVacuum.home,
                           configuration := "Unit1.Em5.Config".cmCathodeAlignTableSuctionPlateVacuum,
                           moduleInterface := "Unit1.Em5.HmiInterface".cmCathodeAlignTableSuctionPlateVacuum,
                           controlNode := "Unit1.Em5.ControlNodes".cmCathodeAlignTableSuctionPlateVacuum);
   "BA030AZSBK32.07" := #instCmCathodeAlignTableSuctionPlateVacuum.goToHomePos AND NOT #statUnitStatus.specialFunctions.dryRun;
   "BA030AZSBK32.06" := #instCmCathodeAlignTableSuctionPlateVacuum.goToWorkPos AND NOT #statUnitStatus.specialFunctions.dryRun;
END_REGION

REGION Network 239: CmCathodeGlassCleaning Home
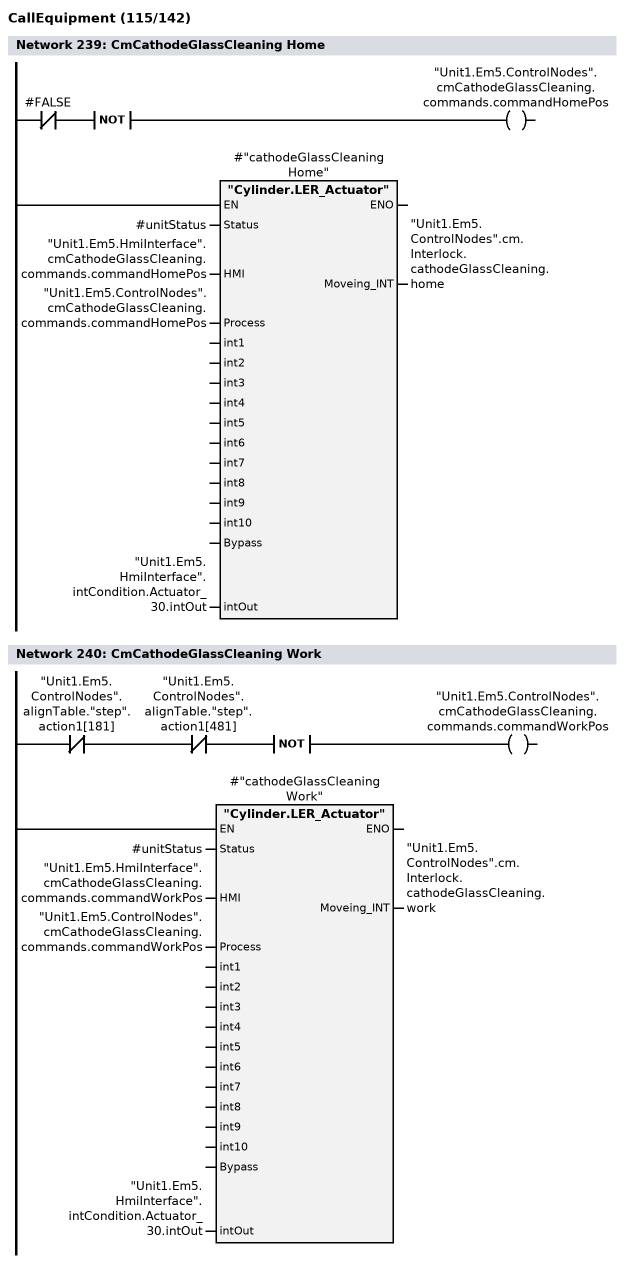
   RUNG wire#powerrail
      I_Contact( #FALSE )
      Not()
      Coil( "Unit1.Em5.ControlNodes".cmCathodeGlassCleaning.commands.commandHomePos )
   END_RUNG
   RUNG wire#powerrail
      #"cathodeGlassCleaning Home"(Status := #unitStatus, HMI := "Unit1.Em5.HmiInterface".cmCathodeGlassCleaning.commands.commandHomePos, Process := "Unit1.Em5.ControlNodes".cmCathodeGlassCleaning.commands.commandHomePos, int1 :=, int2 :=, int3 :=, int4 :=, int5 :=, int6 :=, int7 :=, int8 :=, int9 :=, int10 :=, Bypass :=, intOut := "Unit1.Em5.HmiInterface".intCondition.Actuator_30.intOut, Moveing_INT => "Unit1.Em5.ControlNodes".cm.Interlock.cathodeGlassCleaning.home)
   END_RUNG
   // the same network as SCL:
   "Unit1.Em5.ControlNodes".cmCathodeGlassCleaning.commands.commandHomePos := NOT (NOT #FALSE);
   #"cathodeGlassCleaning Home"(Status := #unitStatus,   // "Cylinder.LER_Actuator"
                           HMI := "Unit1.Em5.HmiInterface".cmCathodeGlassCleaning.commands.commandHomePos,
                           Process := "Unit1.Em5.ControlNodes".cmCathodeGlassCleaning.commands.commandHomePos,
                           intOut := "Unit1.Em5.HmiInterface".intCondition.Actuator_30.intOut,
                           Moveing_INT => "Unit1.Em5.ControlNodes".cm.Interlock.cathodeGlassCleaning.home);
END_REGION

REGION Network 240: CmCathodeGlassCleaning Work
   RUNG wire#powerrail
      I_Contact( "Unit1.Em5.ControlNodes".alignTable."step".action1[181] )
      I_Contact( "Unit1.Em5.ControlNodes".alignTable."step".action1[481] )
      Not()
      Coil( "Unit1.Em5.ControlNodes".cmCathodeGlassCleaning.commands.commandWorkPos )
   END_RUNG
   RUNG wire#powerrail
      #"cathodeGlassCleaning Work"(Status := #unitStatus, HMI := "Unit1.Em5.HmiInterface".cmCathodeGlassCleaning.commands.commandWorkPos, Process := "Unit1.Em5.ControlNodes".cmCathodeGlassCleaning.commands.commandWorkPos, int1 :=, int2 :=, int3 :=, int4 :=, int5 :=, int6 :=, int7 :=, int8 :=, int9 :=, int10 :=, Bypass :=, intOut := "Unit1.Em5.HmiInterface".intCondition.Actuator_30.intOut, Moveing_INT => "Unit1.Em5.ControlNodes".cm.Interlock.cathodeGlassCleaning.work)
   END_RUNG
   // the same network as SCL:
   "Unit1.Em5.ControlNodes".cmCathodeGlassCleaning.commands.commandWorkPos := NOT (NOT "Unit1.Em5.ControlNodes".alignTable."step".action1[181] AND NOT "Unit1.Em5.ControlNodes".alignTable."step".action1[481]);
   #"cathodeGlassCleaning Work"(Status := #unitStatus,   // "Cylinder.LER_Actuator"
                           HMI := "Unit1.Em5.HmiInterface".cmCathodeGlassCleaning.commands.commandWorkPos,
                           Process := "Unit1.Em5.ControlNodes".cmCathodeGlassCleaning.commands.commandWorkPos,
                           intOut := "Unit1.Em5.HmiInterface".intCondition.Actuator_30.intOut,
                           Moveing_INT => "Unit1.Em5.ControlNodes".cm.Interlock.cathodeGlassCleaning.work);
END_REGION

REGION Network 241: Call instCmCathodeGlassCleaning
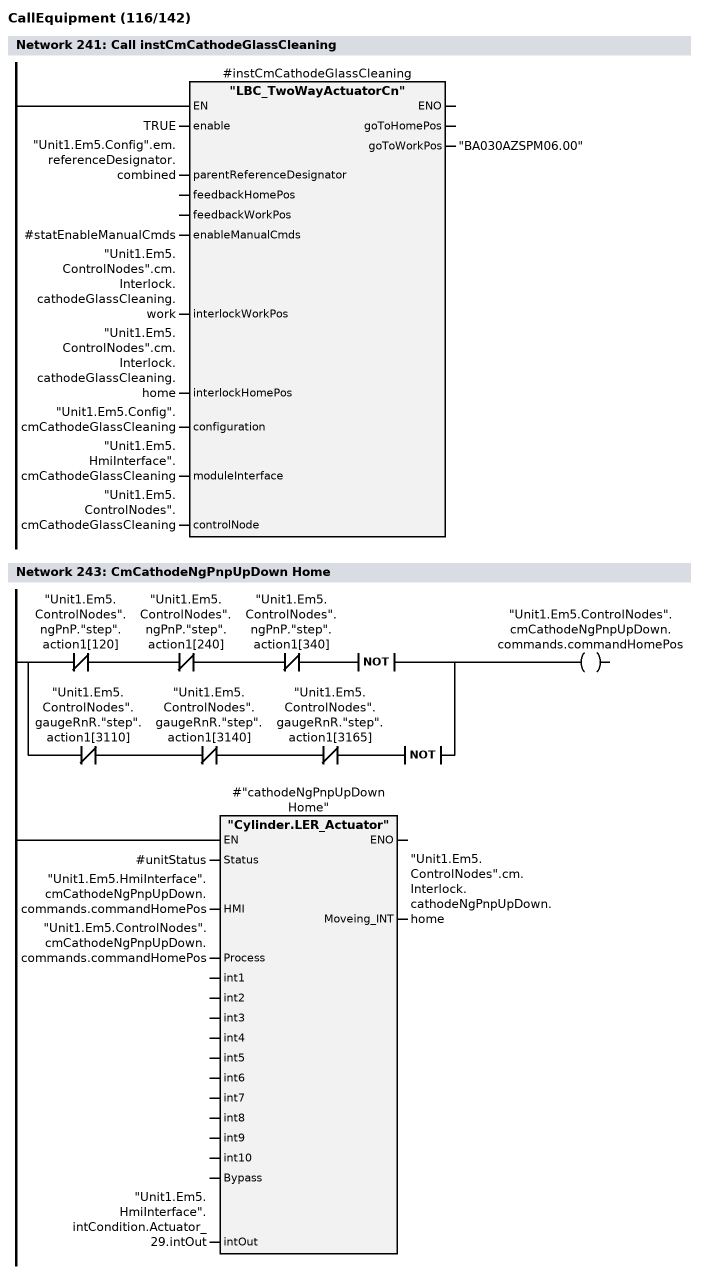
   RUNG wire#powerrail
      #instCmCathodeGlassCleaning(enable := TRUE, parentReferenceDesignator := "Unit1.Em5.Config".em.referenceDesignator.combined, feedbackHomePos :=, feedbackWorkPos :=, enableManualCmds := #statEnableManualCmds, interlockWorkPos := "Unit1.Em5.ControlNodes".cm.Interlock.cathodeGlassCleaning.work, interlockHomePos := "Unit1.Em5.ControlNodes".cm.Interlock.cathodeGlassCleaning.home, configuration := "Unit1.Em5.Config".cmCathodeGlassCleaning, moduleInterface := "Unit1.Em5.HmiInterface".cmCathodeGlassCleaning, controlNode := "Unit1.Em5.ControlNodes".cmCathodeGlassCleaning, goToHomePos =>, goToWorkPos => "BA030AZSPM06.00")
   END_RUNG
   // the same network as SCL:
   #instCmCathodeGlassCleaning(enable := TRUE,   // "LBC_TwoWayActuatorCn"
                           parentReferenceDesignator := "Unit1.Em5.Config".em.referenceDesignator.combined,
                           enableManualCmds := #statEnableManualCmds,
                           interlockWorkPos := "Unit1.Em5.ControlNodes".cm.Interlock.cathodeGlassCleaning.work,
                           interlockHomePos := "Unit1.Em5.ControlNodes".cm.Interlock.cathodeGlassCleaning.home,
                           configuration := "Unit1.Em5.Config".cmCathodeGlassCleaning,
                           moduleInterface := "Unit1.Em5.HmiInterface".cmCathodeGlassCleaning,
                           controlNode := "Unit1.Em5.ControlNodes".cmCathodeGlassCleaning,
                           goToWorkPos => "BA030AZSPM06.00");
END_REGION

REGION Network 243: CmCathodeNgPnpUpDown Home
   RUNG wire#powerrail
      I_Contact( "Unit1.Em5.ControlNodes".ngPnP."step".action1[120] )
      I_Contact( "Unit1.Em5.ControlNodes".ngPnP."step".action1[240] )
      I_Contact( "Unit1.Em5.ControlNodes".ngPnP."step".action1[340] )
      Not()
      wire#w1
      Coil( "Unit1.Em5.ControlNodes".cmCathodeNgPnpUpDown.commands.commandHomePos )
   END_RUNG
   RUNG wire#powerrail
      I_Contact( "Unit1.Em5.ControlNodes".gaugeRnR."step".action1[3110] )
      I_Contact( "Unit1.Em5.ControlNodes".gaugeRnR."step".action1[3140] )
      I_Contact( "Unit1.Em5.ControlNodes".gaugeRnR."step".action1[3165] )
      Not()
   END_RUNG wire#w1
   RUNG wire#powerrail
      #"cathodeNgPnpUpDown Home"(Status := #unitStatus, HMI := "Unit1.Em5.HmiInterface".cmCathodeNgPnpUpDown.commands.commandHomePos, Process := "Unit1.Em5.ControlNodes".cmCathodeNgPnpUpDown.commands.commandHomePos, int1 :=, int2 :=, int3 :=, int4 :=, int5 :=, int6 :=, int7 :=, int8 :=, int9 :=, int10 :=, Bypass :=, intOut := "Unit1.Em5.HmiInterface".intCondition.Actuator_29.intOut, Moveing_INT => "Unit1.Em5.ControlNodes".cm.Interlock.cathodeNgPnpUpDown.home)
   END_RUNG
   // the same network as SCL:
   "Unit1.Em5.ControlNodes".cmCathodeNgPnpUpDown.commands.commandHomePos := NOT (NOT "Unit1.Em5.ControlNodes".ngPnP."step".action1[120] AND NOT "Unit1.Em5.ControlNodes".ngPnP."step".action1[240] AND NOT "Unit1.Em5.ControlNodes".ngPnP."step".action1[340]) OR NOT (NOT "Unit1.Em5.ControlNodes".gaugeRnR."step".action1[3110] AND NOT "Unit1.Em5.ControlNodes".gaugeRnR."step".action1[3140] AND NOT "Unit1.Em5.ControlNodes".gaugeRnR."step".action1[3165]);
   #"cathodeNgPnpUpDown Home"(Status := #unitStatus,   // "Cylinder.LER_Actuator"
                           HMI := "Unit1.Em5.HmiInterface".cmCathodeNgPnpUpDown.commands.commandHomePos,
                           Process := "Unit1.Em5.ControlNodes".cmCathodeNgPnpUpDown.commands.commandHomePos,
                           intOut := "Unit1.Em5.HmiInterface".intCondition.Actuator_29.intOut,
                           Moveing_INT => "Unit1.Em5.ControlNodes".cm.Interlock.cathodeNgPnpUpDown.home);
END_REGION

REGION Network 244: CmCathodeNgPnpUpDown Work
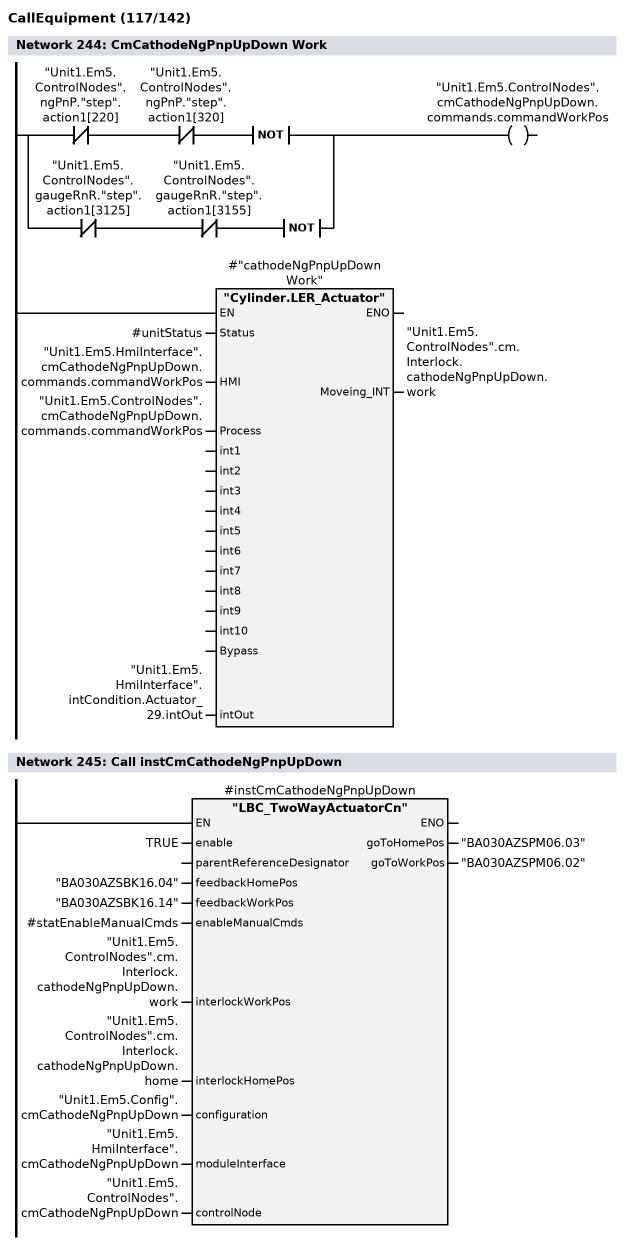
   RUNG wire#powerrail
      I_Contact( "Unit1.Em5.ControlNodes".ngPnP."step".action1[220] )
      I_Contact( "Unit1.Em5.ControlNodes".ngPnP."step".action1[320] )
      Not()
      wire#w1
      Coil( "Unit1.Em5.ControlNodes".cmCathodeNgPnpUpDown.commands.commandWorkPos )
   END_RUNG
   RUNG wire#powerrail
      I_Contact( "Unit1.Em5.ControlNodes".gaugeRnR."step".action1[3125] )
      I_Contact( "Unit1.Em5.ControlNodes".gaugeRnR."step".action1[3155] )
      Not()
   END_RUNG wire#w1
   RUNG wire#powerrail
      #"cathodeNgPnpUpDown Work"(Status := #unitStatus, HMI := "Unit1.Em5.HmiInterface".cmCathodeNgPnpUpDown.commands.commandWorkPos, Process := "Unit1.Em5.ControlNodes".cmCathodeNgPnpUpDown.commands.commandWorkPos, int1 :=, int2 :=, int3 :=, int4 :=, int5 :=, int6 :=, int7 :=, int8 :=, int9 :=, int10 :=, Bypass :=, intOut := "Unit1.Em5.HmiInterface".intCondition.Actuator_29.intOut, Moveing_INT => "Unit1.Em5.ControlNodes".cm.Interlock.cathodeNgPnpUpDown.work)
   END_RUNG
   // the same network as SCL:
   "Unit1.Em5.ControlNodes".cmCathodeNgPnpUpDown.commands.commandWorkPos := NOT (NOT "Unit1.Em5.ControlNodes".ngPnP."step".action1[220] AND NOT "Unit1.Em5.ControlNodes".ngPnP."step".action1[320]) OR NOT (NOT "Unit1.Em5.ControlNodes".gaugeRnR."step".action1[3125] AND NOT "Unit1.Em5.ControlNodes".gaugeRnR."step".action1[3155]);
   #"cathodeNgPnpUpDown Work"(Status := #unitStatus,   // "Cylinder.LER_Actuator"
                           HMI := "Unit1.Em5.HmiInterface".cmCathodeNgPnpUpDown.commands.commandWorkPos,
                           Process := "Unit1.Em5.ControlNodes".cmCathodeNgPnpUpDown.commands.commandWorkPos,
                           intOut := "Unit1.Em5.HmiInterface".intCondition.Actuator_29.intOut,
                           Moveing_INT => "Unit1.Em5.ControlNodes".cm.Interlock.cathodeNgPnpUpDown.work);
END_REGION

REGION Network 245: Call instCmCathodeNgPnpUpDown
   RUNG wire#powerrail
      #instCmCathodeNgPnpUpDown(enable := TRUE, parentReferenceDesignator :=, feedbackHomePos := "BA030AZSBK16.04", feedbackWorkPos := "BA030AZSBK16.14", enableManualCmds := #statEnableManualCmds, interlockWorkPos := "Unit1.Em5.ControlNodes".cm.Interlock.cathodeNgPnpUpDown.work, interlockHomePos := "Unit1.Em5.ControlNodes".cm.Interlock.cathodeNgPnpUpDown.home, configuration := "Unit1.Em5.Config".cmCathodeNgPnpUpDown, moduleInterface := "Unit1.Em5.HmiInterface".cmCathodeNgPnpUpDown, controlNode := "Unit1.Em5.ControlNodes".cmCathodeNgPnpUpDown, goToHomePos => "BA030AZSPM06.03", goToWorkPos => "BA030AZSPM06.02")
   END_RUNG
   // the same network as SCL:
   #instCmCathodeNgPnpUpDown(enable := TRUE,   // "LBC_TwoWayActuatorCn"
                           feedbackHomePos := "BA030AZSBK16.04",
                           feedbackWorkPos := "BA030AZSBK16.14",
                           enableManualCmds := #statEnableManualCmds,
                           interlockWorkPos := "Unit1.Em5.ControlNodes".cm.Interlock.cathodeNgPnpUpDown.work,
                           interlockHomePos := "Unit1.Em5.ControlNodes".cm.Interlock.cathodeNgPnpUpDown.home,
                           configuration := "Unit1.Em5.Config".cmCathodeNgPnpUpDown,
                           moduleInterface := "Unit1.Em5.HmiInterface".cmCathodeNgPnpUpDown,
                           controlNode := "Unit1.Em5.ControlNodes".cmCathodeNgPnpUpDown,
                           goToHomePos => "BA030AZSPM06.03",
                           goToWorkPos => "BA030AZSPM06.02");
END_REGION

REGION Network 247: CmCathodeNgPnp1stFwdBwd Home
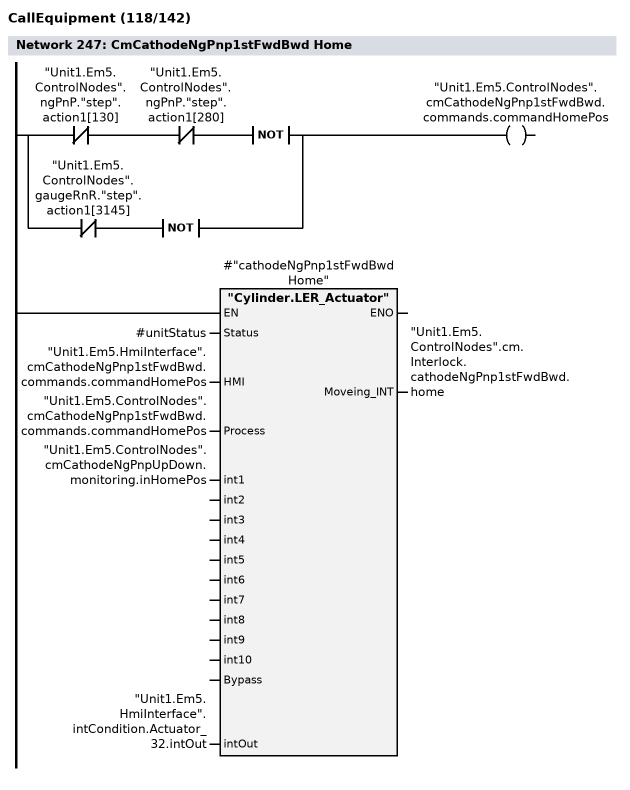
   RUNG wire#powerrail
      I_Contact( "Unit1.Em5.ControlNodes".ngPnP."step".action1[130] )
      I_Contact( "Unit1.Em5.ControlNodes".ngPnP."step".action1[280] )
      Not()
      wire#w1
      Coil( "Unit1.Em5.ControlNodes".cmCathodeNgPnp1stFwdBwd.commands.commandHomePos )
   END_RUNG
   RUNG wire#powerrail
      I_Contact( "Unit1.Em5.ControlNodes".gaugeRnR."step".action1[3145] )
      Not()
   END_RUNG wire#w1
   RUNG wire#powerrail
      #"cathodeNgPnp1stFwdBwd Home"(Status := #unitStatus, HMI := "Unit1.Em5.HmiInterface".cmCathodeNgPnp1stFwdBwd.commands.commandHomePos, Process := "Unit1.Em5.ControlNodes".cmCathodeNgPnp1stFwdBwd.commands.commandHomePos, int1 := "Unit1.Em5.ControlNodes".cmCathodeNgPnpUpDown.monitoring.inHomePos, int2 :=, int3 :=, int4 :=, int5 :=, int6 :=, int7 :=, int8 :=, int9 :=, int10 :=, Bypass :=, intOut := "Unit1.Em5.HmiInterface".intCondition.Actuator_32.intOut, Moveing_INT => "Unit1.Em5.ControlNodes".cm.Interlock.cathodeNgPnp1stFwdBwd.home)
   END_RUNG
   // the same network as SCL:
   "Unit1.Em5.ControlNodes".cmCathodeNgPnp1stFwdBwd.commands.commandHomePos := NOT (NOT "Unit1.Em5.ControlNodes".ngPnP."step".action1[130] AND NOT "Unit1.Em5.ControlNodes".ngPnP."step".action1[280]) OR NOT (NOT "Unit1.Em5.ControlNodes".gaugeRnR."step".action1[3145]);
   #"cathodeNgPnp1stFwdBwd Home"(Status := #unitStatus,   // "Cylinder.LER_Actuator"
                           HMI := "Unit1.Em5.HmiInterface".cmCathodeNgPnp1stFwdBwd.commands.commandHomePos,
                           Process := "Unit1.Em5.ControlNodes".cmCathodeNgPnp1stFwdBwd.commands.commandHomePos,
                           int1 := "Unit1.Em5.ControlNodes".cmCathodeNgPnpUpDown.monitoring.inHomePos,
                           intOut := "Unit1.Em5.HmiInterface".intCondition.Actuator_32.intOut,
                           Moveing_INT => "Unit1.Em5.ControlNodes".cm.Interlock.cathodeNgPnp1stFwdBwd.home);
END_REGION

REGION Network 248: CmCathodeNgPnp1stFwdBwd Work
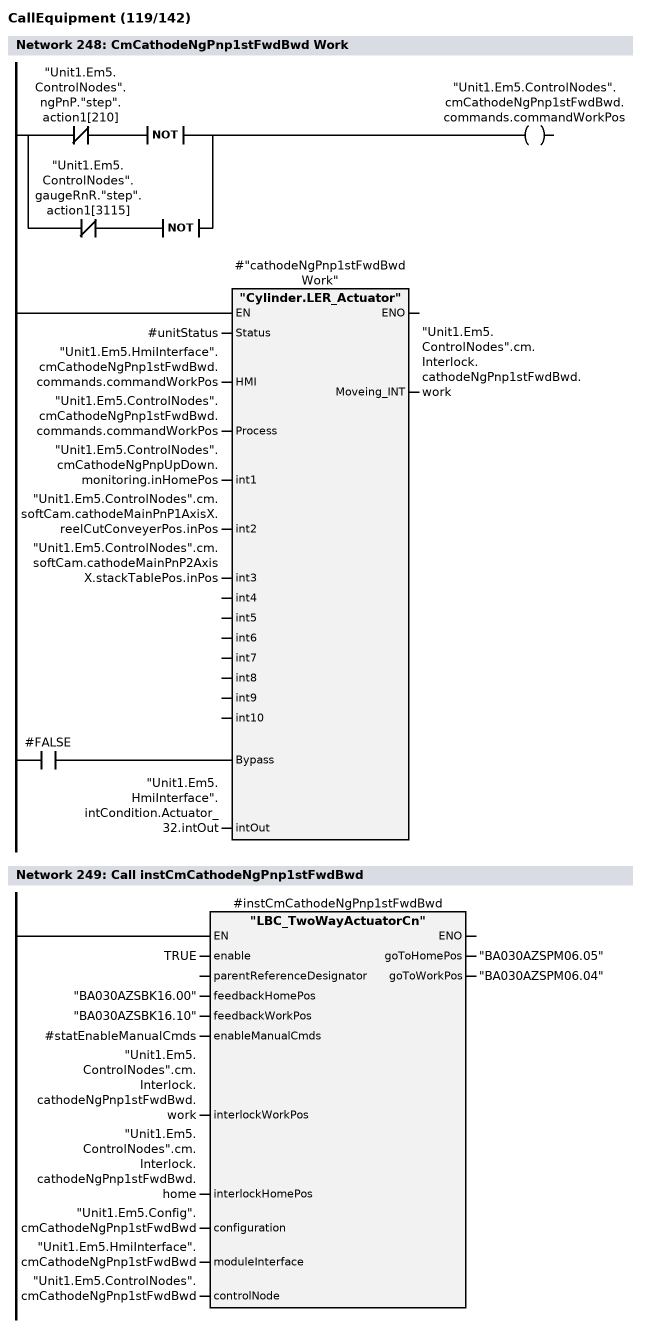
   RUNG wire#powerrail
      I_Contact( "Unit1.Em5.ControlNodes".ngPnP."step".action1[210] )
      Not()
      wire#w1
      Coil( "Unit1.Em5.ControlNodes".cmCathodeNgPnp1stFwdBwd.commands.commandWorkPos )
   END_RUNG
   RUNG wire#powerrail
      I_Contact( "Unit1.Em5.ControlNodes".gaugeRnR."step".action1[3115] )
      Not()
   END_RUNG wire#w1
   RUNG wire#powerrail
      #"cathodeNgPnp1stFwdBwd Work"(Bypass := wire#w2, Status := #unitStatus, HMI := "Unit1.Em5.HmiInterface".cmCathodeNgPnp1stFwdBwd.commands.commandWorkPos, Process := "Unit1.Em5.ControlNodes".cmCathodeNgPnp1stFwdBwd.commands.commandWorkPos, int1 := "Unit1.Em5.ControlNodes".cmCathodeNgPnpUpDown.monitoring.inHomePos, int2 := "Unit1.Em5.ControlNodes".cm.softCam.cathodeMainPnP1AxisX.reelCutConveyerPos.inPos, int3 := "Unit1.Em5.ControlNodes".cm.softCam.cathodeMainPnP2AxisX.stackTablePos.inPos, int4 :=, int5 :=, int6 :=, int7 :=, int8 :=, int9 :=, int10 :=, intOut := "Unit1.Em5.HmiInterface".intCondition.Actuator_32.intOut, Moveing_INT => "Unit1.Em5.ControlNodes".cm.Interlock.cathodeNgPnp1stFwdBwd.work)
   END_RUNG
   RUNG wire#powerrail
      Contact( #FALSE )
   END_RUNG wire#w2
   // the same network as SCL:
   "Unit1.Em5.ControlNodes".cmCathodeNgPnp1stFwdBwd.commands.commandWorkPos := NOT (NOT "Unit1.Em5.ControlNodes".ngPnP."step".action1[210]) OR NOT (NOT "Unit1.Em5.ControlNodes".gaugeRnR."step".action1[3115]);
   #"cathodeNgPnp1stFwdBwd Work"(Status := #unitStatus,   // "Cylinder.LER_Actuator"
                           HMI := "Unit1.Em5.HmiInterface".cmCathodeNgPnp1stFwdBwd.commands.commandWorkPos,
                           Process := "Unit1.Em5.ControlNodes".cmCathodeNgPnp1stFwdBwd.commands.commandWorkPos,
                           int1 := "Unit1.Em5.ControlNodes".cmCathodeNgPnpUpDown.monitoring.inHomePos,
                           int2 := "Unit1.Em5.ControlNodes".cm.softCam.cathodeMainPnP1AxisX.reelCutConveyerPos.inPos,
                           int3 := "Unit1.Em5.ControlNodes".cm.softCam.cathodeMainPnP2AxisX.stackTablePos.inPos,
                           Bypass := #FALSE,
                           intOut := "Unit1.Em5.HmiInterface".intCondition.Actuator_32.intOut,
                           Moveing_INT => "Unit1.Em5.ControlNodes".cm.Interlock.cathodeNgPnp1stFwdBwd.work);
END_REGION

REGION Network 249: Call instCmCathodeNgPnp1stFwdBwd
   RUNG wire#powerrail
      #instCmCathodeNgPnp1stFwdBwd(enable := TRUE, parentReferenceDesignator :=, feedbackHomePos := "BA030AZSBK16.00", feedbackWorkPos := "BA030AZSBK16.10", enableManualCmds := #statEnableManualCmds, interlockWorkPos := "Unit1.Em5.ControlNodes".cm.Interlock.cathodeNgPnp1stFwdBwd.work, interlockHomePos := "Unit1.Em5.ControlNodes".cm.Interlock.cathodeNgPnp1stFwdBwd.home, configuration := "Unit1.Em5.Config".cmCathodeNgPnp1stFwdBwd, moduleInterface := "Unit1.Em5.HmiInterface".cmCathodeNgPnp1stFwdBwd, controlNode := "Unit1.Em5.ControlNodes".cmCathodeNgPnp1stFwdBwd, goToHomePos => "BA030AZSPM06.05", goToWorkPos => "BA030AZSPM06.04")
   END_RUNG
   // the same network as SCL:
   #instCmCathodeNgPnp1stFwdBwd(enable := TRUE,   // "LBC_TwoWayActuatorCn"
                           feedbackHomePos := "BA030AZSBK16.00",
                           feedbackWorkPos := "BA030AZSBK16.10",
                           enableManualCmds := #statEnableManualCmds,
                           interlockWorkPos := "Unit1.Em5.ControlNodes".cm.Interlock.cathodeNgPnp1stFwdBwd.work,
                           interlockHomePos := "Unit1.Em5.ControlNodes".cm.Interlock.cathodeNgPnp1stFwdBwd.home,
                           configuration := "Unit1.Em5.Config".cmCathodeNgPnp1stFwdBwd,
                           moduleInterface := "Unit1.Em5.HmiInterface".cmCathodeNgPnp1stFwdBwd,
                           controlNode := "Unit1.Em5.ControlNodes".cmCathodeNgPnp1stFwdBwd,
                           goToHomePos => "BA030AZSPM06.05",
                           goToWorkPos => "BA030AZSPM06.04");
END_REGION

REGION Network 251: CmCathodeNgPnp2ndFwdBwd Home
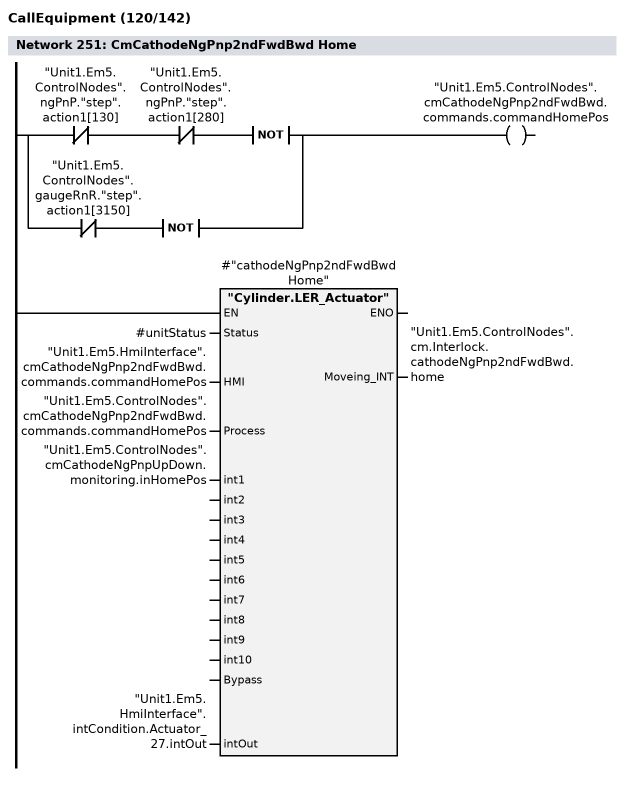
   RUNG wire#powerrail
      I_Contact( "Unit1.Em5.ControlNodes".ngPnP."step".action1[130] )
      I_Contact( "Unit1.Em5.ControlNodes".ngPnP."step".action1[280] )
      Not()
      wire#w1
      Coil( "Unit1.Em5.ControlNodes".cmCathodeNgPnp2ndFwdBwd.commands.commandHomePos )
   END_RUNG
   RUNG wire#powerrail
      I_Contact( "Unit1.Em5.ControlNodes".gaugeRnR."step".action1[3150] )
      Not()
   END_RUNG wire#w1
   RUNG wire#powerrail
      #"cathodeNgPnp2ndFwdBwd Home"(Status := #unitStatus, HMI := "Unit1.Em5.HmiInterface".cmCathodeNgPnp2ndFwdBwd.commands.commandHomePos, Process := "Unit1.Em5.ControlNodes".cmCathodeNgPnp2ndFwdBwd.commands.commandHomePos, int1 := "Unit1.Em5.ControlNodes".cmCathodeNgPnpUpDown.monitoring.inHomePos, int2 :=, int3 :=, int4 :=, int5 :=, int6 :=, int7 :=, int8 :=, int9 :=, int10 :=, Bypass :=, intOut := "Unit1.Em5.HmiInterface".intCondition.Actuator_27.intOut, Moveing_INT => "Unit1.Em5.ControlNodes".cm.Interlock.cathodeNgPnp2ndFwdBwd.home)
   END_RUNG
   // the same network as SCL:
   "Unit1.Em5.ControlNodes".cmCathodeNgPnp2ndFwdBwd.commands.commandHomePos := NOT (NOT "Unit1.Em5.ControlNodes".ngPnP."step".action1[130] AND NOT "Unit1.Em5.ControlNodes".ngPnP."step".action1[280]) OR NOT (NOT "Unit1.Em5.ControlNodes".gaugeRnR."step".action1[3150]);
   #"cathodeNgPnp2ndFwdBwd Home"(Status := #unitStatus,   // "Cylinder.LER_Actuator"
                           HMI := "Unit1.Em5.HmiInterface".cmCathodeNgPnp2ndFwdBwd.commands.commandHomePos,
                           Process := "Unit1.Em5.ControlNodes".cmCathodeNgPnp2ndFwdBwd.commands.commandHomePos,
                           int1 := "Unit1.Em5.ControlNodes".cmCathodeNgPnpUpDown.monitoring.inHomePos,
                           intOut := "Unit1.Em5.HmiInterface".intCondition.Actuator_27.intOut,
                           Moveing_INT => "Unit1.Em5.ControlNodes".cm.Interlock.cathodeNgPnp2ndFwdBwd.home);
END_REGION

REGION Network 252: CmCathodeNgPnp2ndFwdBwd Work
